   (*Предупреждение. Неисправность датчика Давления газа перед горелкой*)
   IF "P_gas_before_burner".N_module <> 0 AND "Warning_Enable".Sensor_P_gas_before_burner THEN
       "Warning".Sensor_P_gas_before_burner := "P_gas_before_burner".Error_sensor;
   ELSE
       "Warning".Sensor_P_gas_before_burner := FALSE;
   END_IF;

   (*Предупреждение. Неисправность датчика Давления воздуха к горелке*)
   IF "P_air_burner".N_module <> 0 AND "Warning_Enable".Sensor_P_air_burner THEN
       "Warning".Sensor_P_air_burner := "P_air_burner".Error_sensor;
   ELSE
       "Warning".Sensor_P_air_burner := FALSE;
   END_IF;

   (*Предупреждение. Неисправность датчика Положения рег. заслонки питательной воды на котел*)
   IF "ZRW_position".N_module <> 0 AND "Warning_Enable".Sensor_ZRW_position THEN
       "Warning".Sensor_ZRW_position := "ZRW_position".Error_sensor;
   ELSE
       "Warning".Sensor_ZRW_position := FALSE;
   END_IF;

   (*Предупреждение. Неисправность датчика Положения рег. заслонки газа перед котлом*)
   IF "ZRG_position".N_module <> 0 AND "Warning_Enable".Sensor_ZRG_position THEN
       "Warning".Sensor_ZRG_position := "ZRG_position".Error_sensor;
   ELSE
       "Warning".Sensor_ZRG_position := FALSE;
   END_IF;

   (*Предупреждение. Неисправность датчика Положения направл. аппарата вентилятора*)
   IF "NAV_position".N_module <> 0 AND "Warning_Enable".Sensor_NAV_position THEN
       "Warning".Sensor_NAV_position := "NAV_position".Error_sensor;
   ELSE
       "Warning".Sensor_NAV_position := FALSE;
   END_IF;

   (*Предупреждение. Неисправность датчика Положения направл. аппарата дымососа*)
   IF "NAD_position".N_module <> 0 AND "Warning_Enable".Sensor_NAD_position THEN
       "Warning".Sensor_NAD_position := "NAD_position".Error_sensor;
   ELSE
       "Warning".Sensor_NAD_position := FALSE;
   END_IF;

   (*Предупреждение. Неисправность датчика Температуры уходящих дымовых газов  перед экономайзером*)
   IF "T_exhaust_gas_before_economizer".N_module <> 0 AND "Warning_Enable".Sensor_T_exhaust_gas_before_economizer THEN
       "Warning".Sensor_T_exhaust_gas_before_economizer := "T_exhaust_gas_before_economizer".Error_sensor;
   ELSE
       "Warning".Sensor_T_exhaust_gas_before_economizer := FALSE;
   END_IF;

   (*Предупреждение. Неисправность датчика Температуры уходящих дымовых газов  после экономайзера*)
   IF "T_exhaust_gas_after_economizer".N_module <> 0 AND "Warning_Enable".Sensor_T_exhaust_gas_after_economizer THEN
       "Warning".Sensor_T_exhaust_gas_after_economizer := "T_exhaust_gas_after_economizer".Error_sensor;
   ELSE
       "Warning".Sensor_T_exhaust_gas_after_economizer := FALSE;
   END_IF;

   (*Предупреждение. Неисправность датчика Разрежения в дымоходе перед экономайзером*)
   IF "dP_exhaust_gas_before_economizer".N_module <> 0 AND "Warning_Enable".Sensor_dP_exhaust_gas_before_economizer THEN
       "Warning".Sensor_dP_exhaust_gas_before_economizer := "dP_exhaust_gas_before_economizer".Error_sensor;
   ELSE
       "Warning".Sensor_dP_exhaust_gas_before_economizer := FALSE;
   END_IF;

   (*Предупреждение. Неисправность датчика Разрежения в дымоходе после экономайзера*)
   IF "dP_exhaust_gas_after_economizer".N_module <> 0 AND "Warning_Enable".Sensor_dP_exhaust_gas_after_economizer THEN
       "Warning".Sensor_dP_exhaust_gas_after_economizer := "dP_exhaust_gas_after_economizer".Error_sensor;
   ELSE
       "Warning".Sensor_dP_exhaust_gas_after_economizer := FALSE;
   END_IF;

   (*Предупреждение. Неисправность датчика Уровня воды в барабане*)
   IF "L_water".N_module <> 0 AND "Warning_Enable".Sensor_L_water THEN
       "Warning".Sensor_L_water := "L_water".Error_sensor;
   ELSE
       "Warning".Sensor_L_water := FALSE;
   END_IF;

   (*Предупреждение. Неисправность датчика Давления газа перед БГ*)
   IF "P_gas_before_BG".N_module <> 0 AND "Warning_Enable".Sensor_P_gas_before_BG THEN
       "Warning".Sensor_P_gas_before_BG := "P_gas_before_BG".Error_sensor;
   ELSE
       "Warning".Sensor_P_gas_before_BG := FALSE;
   END_IF;

   (*Предупреждение. Неисправность датчика Температуры газа перед БГ*)
   IF "T_gas_before_BG".N_module <> 0 AND "Warning_Enable".Sensor_T_gas_before_BG THEN
       "Warning".Sensor_T_gas_before_BG := "T_gas_before_BG".Error_sensor;
   ELSE
       "Warning".Sensor_T_gas_before_BG := FALSE;
   END_IF;

   (*Предупреждение. Неисправность датчика Давления пара в магистраль*)
   IF "P_steam_pipe".N_module <> 0 AND "Warning_Enable".Sensor_P_steam_pipe THEN
       "Warning".Sensor_P_steam_pipe := "P_steam_pipe".Error_sensor;
   ELSE
       "Warning".Sensor_P_steam_pipe := FALSE;
   END_IF;

   (*Предупреждение. Неисправность датчика Температуры пара в магистраль*)
   IF "T_steam".N_module <> 0 AND "Warning_Enable".Sensor_T_steam THEN
       "Warning".Sensor_T_steam := "T_steam".Error_sensor;
   ELSE
       "Warning".Sensor_T_steam := FALSE;
   END_IF;

   (*Предупреждение. Неисправность датчика Текущего значение частоты ПЧ вентилятора*)
   IF "DV_current_frequency".N_module <> 0 AND "Warning_Enable".Sensor_DV_current_frequency THEN
       "Warning".Sensor_DV_current_frequency := "DV_current_frequency".Error_sensor;
   ELSE
       "Warning".Sensor_DV_current_frequency := FALSE;
   END_IF;

   (*Предупреждение. Неисправность датчика Текущего значение частоты ПЧ дымососа*)
   IF "DS_current_frequency".N_module <> 0 AND "Warning_Enable".Sensor_DS_current_frequency THEN
       "Warning".Sensor_DS_current_frequency := "DS_current_frequency".Error_sensor;
   ELSE
       "Warning".Sensor_DS_current_frequency := FALSE;
   END_IF;

   (*Предупреждение. Сработал ограничитель крутящего момента ЗДСВ перед котлом*)
   "Warning_Timer".warning_9_PT := T_CONV(INT_TO_DINT(5) * 1000);
   IF "ZDSV_before_boiler_limit_rotational_moment".Enable AND "Warning_Enable".ZDSV_before_boiler_limit_rotational_moment THEN
       "Warning_Timer".warning_9_IN := "ZDSV_before_boiler_limit_rotational_moment".Value;
       "Warning".ZDSV_before_boiler_limit_rotational_moment := "Warning_Timer".warning_9_Q;
   ELSE
       "Warning_Timer".warning_9_IN := FALSE;
       "Warning".ZDSV_before_boiler_limit_rotational_moment := FALSE;
   END_IF;

   (*Предупреждение. Сработал ограничитель крутящего момента ГПЗ*)
   "Warning_Timer".warning_10_PT := T_CONV(INT_TO_DINT(5) * 1000);
   IF "GPZ_limit_rotational_moment".Enable AND "Warning_Enable".GPZ_limit_rotational_moment THEN
       "Warning_Timer".warning_10_IN := "GPZ_limit_rotational_moment".Value;
       "Warning".GPZ_limit_rotational_moment := "Warning_Timer".warning_10_Q;
   ELSE
       "Warning_Timer".warning_10_IN := FALSE;
       "Warning".GPZ_limit_rotational_moment := FALSE;
   END_IF;

   (*Предупреждение. Вызов к шакафу электропитания*)
   IF "Call_power_supply_cabinet".N_module<>0 AND "Warning_Enable".Call_power_supply_cabinet THEN
       "Warning".Call_power_supply_cabinet := "Call_power_supply_cabinet".Value;
   ELSE
       "Warning".Call_power_supply_cabinet := FALSE;
   END_IF;

   (*Предупреждение. ДВ. Необходимо включить QF ПЧ*)
   IF "DV_dist_control".Value AND "DV_invertor_mode".Value AND NOT "DV_invertor_QF_on".Value AND "DV_invertor_QF_on".N_module<>0 AND "Warning_Enable".DV_need_on_QF_invertor THEN
       "Warning".DV_need_on_QF_invertor := TRUE;
   ELSE
       "Warning".DV_need_on_QF_invertor := FALSE;
   END_IF;

   (*Предупреждение. ДВ. Необходимо включить QF Сети*)
   IF "DV_dist_control".Value AND "DV_powergrid_mode".Value AND NOT "DV_powergrid_QF_on".Value AND "DV_powergrid_QF_on".N_module<>0 AND "Warning_Enable".DV_need_on_QF_powergrid THEN
       "Warning".DV_need_on_QF_powergrid := TRUE;
   ELSE
       "Warning".DV_need_on_QF_powergrid := FALSE;
   END_IF;

   (*Предупреждение. ДВ. Неисправность напряжения в Сети ШУД*)
   IF "DV_no_voltage".N_module<>0 AND "Warning_Enable".DV_no_voltage THEN
       "Warning".DV_no_voltage := "DV_no_voltage".Value;
   ELSE
       "Warning".DV_no_voltage := FALSE;
   END_IF;

   (*Предупреждение. ДС. Необходимо включить QF ПЧ*)
   IF "DS_dist_control".Value AND "DS_invertor_mode".Value AND NOT "DS_invertor_QF_on".Value AND "DS_invertor_QF_on".N_module<>0 AND "Warning_Enable".DS_need_on_QF_invertor THEN
       "Warning".DS_need_on_QF_invertor := TRUE;
   ELSE
       "Warning".DS_need_on_QF_invertor := FALSE;
   END_IF;

   (*Предупреждение. ДС. Необходимо включить QF Сети*)
   IF "DS_dist_control".Value AND "DS_powergrid_mode".Value AND NOT "DS_powergrid_QF_on".Value AND "DS_powergrid_QF_on".N_module<>0 AND "Warning_Enable".DS_need_on_QF_powergrid THEN
       "Warning".DS_need_on_QF_powergrid := TRUE;
   ELSE
       "Warning".DS_need_on_QF_powergrid := FALSE;
   END_IF;

   (*Предупреждение. ДС. Неисправность напряжения в Сети ШУД*)
   IF "DS_no_voltage".N_module<>0 AND "Warning_Enable".DS_no_voltage THEN
       "Warning".DS_no_voltage := "DS_no_voltage".Value;
   ELSE
       "Warning".DS_no_voltage := FALSE;
   END_IF;

   (*Предупреждение. Нет питания ШЭУ*)
   IF "SHEU_voltage_ok".N_module<>0 AND "Warning_Enable".SHEU_no_voltage THEN
       "Warning".SHEU_no_voltage := NOT "SHEU_voltage_ok".Value;
   ELSE
       "Warning".SHEU_no_voltage := FALSE;
   END_IF;

   (*Предупреждение. Питание контроллера от ИБП*)
   IF "Power_PLC_from_UPS".N_module<>0 AND "Warning_Enable".Power_PLC_from_UPS THEN
       "Warning".Power_PLC_from_UPS := "Power_PLC_from_UPS".Value;
   ELSE
       "Warning".Power_PLC_from_UPS := FALSE;
   END_IF;

   (*Предупреждение. Низкий заряд батареи ИБП*)
   IF "UPS_Low_charge".N_module<>0 AND "Warning_Enable".UPS_Low_charge THEN
       "Warning".UPS_Low_charge := "UPS_Low_charge".Value;
   ELSE
       "Warning".UPS_Low_charge := FALSE;
   END_IF;

   (*Предупреждение. Нет питания ЗРГ*)
   IF "ZRG_voltage_ok".N_module<>0 AND "Warning_Enable".ZRG_no_voltage THEN
       "Warning".ZRG_no_voltage := NOT "ZRG_voltage_ok".Value;
   ELSE
       "Warning".ZRG_no_voltage := FALSE;
   END_IF;

   (*Предупреждение. Нет питания ЗДГ*)
   IF "ZDG_voltage_ok".N_module<>0 AND "Warning_Enable".ZDG_no_voltage THEN
       "Warning".ZDG_no_voltage := NOT "ZDG_voltage_ok".Value;
   ELSE
       "Warning".ZDG_no_voltage := FALSE;
   END_IF;

   (*Предупреждение. Нет питания НАВ*)
   IF "NAV_voltage_ok".N_module<>0 AND "Warning_Enable".NAV_no_voltage THEN
       "Warning".NAV_no_voltage := NOT "NAV_voltage_ok".Value;
   ELSE
       "Warning".NAV_no_voltage := FALSE;
   END_IF;

   (*Предупреждение. Нет питания НАД*)
   IF "NAD_voltage_ok".N_module<>0 AND "Warning_Enable".NAD_no_voltage THEN
       "Warning".NAD_no_voltage := NOT "NAD_voltage_ok".Value;
   ELSE
       "Warning".NAD_no_voltage := FALSE;
   END_IF;

   (*Предупреждение. Нет питания ЗДСВ перед котлом*)
   IF "ZDSV_before_boiler_voltage_ok".N_module<>0 AND "Warning_Enable".ZDSV_before_boiler_no_voltage THEN
       "Warning".ZDSV_before_boiler_no_voltage := NOT "ZDSV_before_boiler_voltage_ok".Value;
   ELSE
       "Warning".ZDSV_before_boiler_no_voltage := FALSE;
   END_IF;

   (*Предупреждение. Нет питания ГПЗ*)
   IF "GPZ_voltage_ok".N_module <> 0 AND "Warning_Enable".GPZ_no_voltage THEN
       "Warning".GPZ_no_voltage := NOT "GPZ_voltage_ok".Value;
   ELSE
       "Warning".GPZ_no_voltage := FALSE;
   END_IF;

   (*Предупреждение. Нет питания ЗРВ*)
   IF "ZRW_voltage_ok".N_module <> 0 AND "Warning_Enable".ZRW_no_voltage THEN
       "Warning".ZRW_no_voltage := NOT "ZRW_voltage_ok".Value;
   ELSE
       "Warning".ZRW_no_voltage := FALSE;
   END_IF;

   (*Предупреждение. Авария ПЧ ДВ*)
   IF "DV_Invertor_alarm".N_module<>0 AND "DV_invertor_mode".Value AND "Warning_Enable".DV_invertor_alarm THEN
       "Warning".DV_invertor_alarm := "DV_Invertor_alarm".Value;
   ELSE
       "Warning".DV_invertor_alarm := FALSE;
   END_IF;

   (*Предупреждение. Авария ПЧ ДС*)
   IF "DS_Invertor_alarm".N_module<>0 AND "DS_invertor_mode".Value AND "Warning_Enable".DS_invertor_alarm THEN
       "Warning".DS_invertor_alarm := "DS_Invertor_alarm".Value;
   ELSE
       "Warning".DS_invertor_alarm := FALSE;
   END_IF;

   (*Предупреждение. ЗРГ в местном режиме управления*)
   "Warning".ZRG_manual := "Warning_Enable".ZRG_manual AND NOT "ZRG_avto".Value;

   (*Предупреждение. НАВ в местном режиме управления*)
   "Warning".NAV_manual := "Warning_Enable".NAV_manual AND NOT "NAV_avto".Value;

   (*Предупреждение. НАД в местном режиме управления*)
   "Warning".NAD_manual := "Warning_Enable".NAD_manual AND NOT "NAD_avto".Value;

   (*Предупреждение. ДВ в местном режиме управления*)
   "Warning".DV_manual := "Warning_Enable".DV_manual AND "DV_local_control".Value;

   (*Предупреждение. ДС в местном режиме управления*)
   "Warning".DS_manual := "Warning_Enable".DS_manual AND "DS_local_control".Value;

   (*Предупреждение. ЗРВ в местном режиме управления*)
   "Warning".ZRW_manual := "Warning_Enable".ZRW_manual AND NOT "ZRW_avto".Value;

   (*Пламя запальника потухло*)
   "Warning_Timer".warning_1_PT := T_CONV(INT_TO_DINT("Warning_SP".TIME_Not_flame_Igniter));
   IF "Warning_Enable".Not_flame_Igniter THEN
       "Warning_Timer".warning_1_IN := NOT "Igniter_flame".Value;
       IF "Warning_Timer".warning_1_Q THEN
           "Warning".Not_flame_Igniter := TRUE;
       END_IF;
   ELSE
       "Warning_Timer".warning_1_IN := FALSE;
       //"Warning".Not_flame_Igniter := FALSE;
   END_IF;

   (*ПЗК2 не открылся*)
   "Warning_Timer".warning_2_PT := T_CONV(INT_TO_DINT("Warning_SP".TIME_PZK2_not_open) * 1000);
   IF "Warning_Enable".PZK2_not_open THEN
       "Warning_Timer".warning_2_IN := NOT "PZK2_open".Value;
       IF "Warning_Timer".warning_2_Q THEN
           "Warning".PZK2_not_open := TRUE;
       END_IF;
   ELSE
       "Warning_Timer".warning_2_IN := FALSE;
       //"Warning".PZK2_not_open := FALSE;
   END_IF;

   (*Понижение давления сетевой воды*)
   IF ("P_water_before_regul".Value <"Warning_SP".P_water_min AND NOT"P_water_before_regul".Error_sensor AND "P_water_before_regul".N_module <> 0) THEN
       "Warning".P_water_min := TRUE;
   ELSE
       "Warning".P_water_min := FALSE;
   END_IF;

   (*Понижение уровня воды в барабане*)
   "Warning_Timer".warning_3_PT := T_CONV(INT_TO_DINT("Warning_SP".TIME_L_water_min) * 1000);
   IF "Warning_Enable".L_water_min THEN
       "Warning_Timer".warning_3_IN := "L_water".Value < "Warning_SP".L_water_min AND NOT "L_water".Error_sensor AND "L_water".N_module <> 0;
       "Warning".L_water_min := "Warning_Timer".warning_3_Q;
   ELSE
       "Warning_Timer".warning_3_IN := FALSE;
       "Warning".L_water_min := FALSE;
   END_IF;

   (*Повышение уровня воды в барабане*)
   "Warning_Timer".warning_4_PT := T_CONV(INT_TO_DINT("Warning_SP".TIME_L_water_max) * 1000);
   IF "Warning_Enable".L_water_max THEN
       "Warning_Timer".warning_4_IN := "L_water".Value > "Warning_SP".L_water_max AND NOT "L_water".Error_sensor AND "L_water".N_module <> 0;
       "Warning".L_water_max := "Warning_Timer".warning_4_Q;
   ELSE
       "Warning_Timer".warning_4_IN := FALSE;
       "Warning".L_water_max := FALSE;
   END_IF;

   (*Повышение давления пара в барабане*)
   "Warning_Timer".warning_5_PT := T_CONV(INT_TO_DINT("Warning_SP".TIME_P_steam_max) * 1000);
   IF "Warning_Enable".P_steam_max THEN
       "Warning_Timer".warning_5_IN := "P_steam".Value > "Warning_SP".P_steam_max AND NOT "P_steam".Error_sensor AND "P_steam".N_module <> 0;
       "Warning".P_steam_max := "Warning_Timer".warning_5_Q;
   ELSE
       "Warning_Timer".warning_5_IN := FALSE;
       "Warning".P_steam_max := FALSE;
   END_IF;

   (*СО порог 1*)
   IF "Warning_Enable".CO2 THEN
       "Warning".CO2 := "CO_1".Value;
   ELSE
       "Warning".CO2 := FALSE;
   END_IF;

   (*Предупреждение. Понижение разряжения в топке*)
   "Warning_Timer".warning_6_PT := T_CONV(INT_TO_DINT("Alarm_SP".TIME_dP_furnace_boiler_min) * 1000);
   IF "Technology".Regim = 3 AND ("Technology".Regim_ventilation_step = 23 OR "Technology".Regim_ventilation_step = 24) AND "Warning_Enable".dP_furnace_boiler_min THEN
       "Warning_Timer".warning_6_IN := "dP_furnace_boiler_min".Value OR ("dP_furnace_boiler".Value > "Alarm_SP".dP_furnace_boiler_min AND NOT "dP_furnace_boiler".Error_sensor AND "dP_furnace_boiler".N_module <> 0);
       IF "Warning_Timer".warning_6_Q THEN
           "Warning".dP_furnace_boiler_min := TRUE;
       END_IF;
   ELSE
       "Warning_Timer".warning_6_IN := FALSE;
       "Warning".dP_furnace_boiler_min := FALSE;
   END_IF;

   (*Предупреждение. Понижение давления воздуха перед горелкой *)
   "Warning_Timer".warning_7_PT := T_CONV(INT_TO_DINT("Alarm_SP".TIME_P_air_before_burner_min) * 1000);
   IF "Technology".Regim = 3 AND ("Technology".Regim_ventilation_step = 23 OR "Technology".Regim_ventilation_step = 24) AND "Warning_Enable".P_air_before_burner_min THEN
       "Warning_Timer".warning_7_IN := "P_air_before_burner_min".Value OR ("P_air_burner".Value < "Alarm_SP".P_air_before_burner_min AND NOT "P_air_burner".Error_sensor AND "P_air_burner".N_module<>0);
       IF "Warning_Timer".warning_7_Q THEN
           "Warning".P_air_before_burner_min := TRUE;
       END_IF;
   ELSE
       "Warning_Timer".warning_7_IN := FALSE;
       "Warning".P_air_before_burner_min := FALSE;
   END_IF;

   (*ЗДГ не закрылась*)
   "Warning_Timer".warning_8_PT := T_CONV(INT_TO_DINT("Warning_SP".TIME_ZDG_not_close) * 1000);
   IF "Warning_Enable".ZDG_not_close THEN
       "Warning_Timer".warning_8_IN := "ZDG_no_close".Value;
       IF "Warning_Timer".warning_8_Q THEN
           "Warning".ZDG_not_close := TRUE;
       END_IF;
   ELSE
       "Warning_Timer".warning_8_IN := FALSE;
   END_IF;

   (*Предупреждение. Имеется блокировка защиты *)
   IF "Protections_BLOCK".P_gas_before_BG_max OR
       "Protections_BLOCK".P_gas_before_BG_min OR
       "Protections_BLOCK".P_gas_before_burner_min OR
       "Protections_BLOCK".P_gas_before_burner_max OR
       "Protections_BLOCK".DS_off OR
       "Protections_BLOCK".DV_off OR
       "Protections_BLOCK".dP_in_furnance_min OR
       "Protections_BLOCK".P_air_before_burner_min OR
       "Protections_BLOCK".L_water_min OR
       "Protections_BLOCK".L_water_max OR
       "Protections_BLOCK".P_steam_max OR
       "Protections_BLOCK".Not_flame_burner OR
       "Protections_BLOCK".Alarm_stop_HMI OR
       "Protections_BLOCK".Alarm_stop_SCADA THEN
       "Warning".protection_block := TRUE;
   ELSE
       "Warning".protection_block := FALSE;
   END_IF;

   (*СБРОС аварий для журнала событий*)
   IF "Alarm".Reset_alarms THEN
       "HMI".Reset_alarms_Log := TRUE;
   END_IF;

   (*Сброс всех аварий и предупреждений*)
   IF "Alarm".Reset_alarms = TRUE OR
       "Btn_Sound".Value THEN
       (*Повышение давления газа перед БГ*)
       IF NOT "Alarm_Timer".alarm_1_Q THEN
           "Alarm".P_gas_before_BG_max := FALSE;
       END_IF;
       (*Понижение давления газа перед БГ*)
       IF NOT "Alarm_Timer".alarm_2_Q THEN
           "Alarm".P_gas_before_BG_min := FALSE;
       END_IF;
       (*Понижение давления газа перед горелкой*)
       IF NOT "Alarm_Timer".alarm_3_Q THEN
           "Alarm".P_gas_before_burner_min := FALSE;
       END_IF;
       (*Повышение давления газа перед горелкой*)
       IF NOT "Alarm_Timer".alarm_4_Q THEN
           "Alarm".P_gas_before_burner_max := FALSE;
       END_IF;
       (*Отключение ДС*)
       IF NOT "Alarm_Timer".alarm_5_Q THEN
           "Alarm".DS_off := FALSE;
       END_IF;
       (*Отключение ДВ*)
       IF NOT "Alarm_Timer".alarm_6_Q THEN
           "Alarm".DV_off := FALSE;
       END_IF;
       (*Понижение разряжения в топке*)
       IF NOT "Alarm_Timer".alarm_7_Q THEN
           "Alarm".dP_furnace_boiler_min := FALSE;
       END_IF;
       (*Понижение давления воздуха перед горелкой *)
       IF NOT "Alarm_Timer".alarm_8_Q THEN
           "Alarm".P_air_before_burner_min := FALSE;
       END_IF;
       (*Понижение уровня воды в барабане*)
       IF NOT "Alarm_Timer".alarm_9_Q THEN
           "Alarm".L_water_min := FALSE;
       END_IF;
       (*Повышение уровня воды в барабане*)
       IF NOT "Alarm_Timer".alarm_10_Q THEN
           "Alarm".L_water_max := FALSE;
       END_IF;
       (*Повышение давления пара в барабане*)
       IF NOT "Alarm_Timer".alarm_11_Q THEN
           "Alarm".P_steam_max := FALSE;
       END_IF;
       (*Невоспламенение или погасание факела горелки котла*)
       IF NOT "Alarm_Timer".alarm_12_Q THEN
           "Alarm".Not_flame_burner := FALSE;
       END_IF;
       (*Нажата кнопка аварийного останова на панели оператора*)
       "Alarm".Alarm_stop_HMI := FALSE;
       (*Нажата кнопка аварийного останова на SCADA*)
       "Alarm".Alarm_stop_SCADA := FALSE;
       (*СО2 порог 2*)
       IF NOT "Alarm_Timer".alarm_13_Q THEN
           "Alarm".CO2 := FALSE;
       END_IF;
       (*CH4*)
       IF NOT "Alarm_Timer".alarm_14_Q THEN
           "Alarm".CH4 := FALSE;
       END_IF;
       (*Пламя запальника потухло*)
       IF NOT "Warning_Timer".warning_1_Q THEN
           "Warning".Not_flame_Igniter := FALSE;
       END_IF;
       (*ПЗК2 не открылся*)
       IF NOT "Warning_Timer".warning_2_Q THEN
           "Warning".PZK2_not_open := FALSE;
       END_IF;
       (*Понижение уровня воды в барабане*)
       IF NOT "Warning_Timer".warning_3_Q THEN
           "Warning".L_water_min := FALSE;
       END_IF;
       (*Повышение уровня воды в барабане*)
       IF NOT "Warning_Timer".warning_4_Q THEN
           "Warning".L_water_max := FALSE;
       END_IF;
       (*Повышение давления пара в барабане*)
       IF NOT "Warning_Timer".warning_5_Q THEN
           "Warning".P_steam_max := FALSE;
       END_IF;
       (*Предупреждение. Понижение разряжения в топке*)
       IF NOT "Warning_Timer".warning_6_Q THEN
           "Warning".dP_furnace_boiler_min := FALSE;
       END_IF;
       (*Предупреждение. Понижение давления воздуха перед горелкой *)
       IF NOT "Warning_Timer".warning_7_Q THEN
           "Warning".P_air_before_burner_min := FALSE;
       END_IF;
       (*ЗДГ не закрылась*)
       IF NOT "Warning_Timer".warning_8_Q THEN
           "Warning".ZDG_not_close := FALSE;
       END_IF;
       "Alarm".Reset_alarms := FALSE;
   END_IF;

   (*Формирование обобщенного признака аварии*)
   "Alarm".Global_alarm := "Alarm".P_gas_before_BG_max OR
   "Alarm".P_gas_before_BG_min OR
   "Alarm".P_gas_before_burner_min OR
   "Alarm".P_gas_before_burner_max OR
   "Alarm".DS_off OR
   "Alarm".DV_off OR
   "Alarm".dP_furnace_boiler_min OR
   "Alarm".P_air_before_burner_min OR
   "Alarm".L_water_min OR
   "Alarm".L_water_max OR
   "Alarm".P_steam_max OR
   "Alarm".Not_flame_burner OR
   "Alarm".Alarm_stop_HMI OR
   "Alarm".Alarm_stop_SCADA OR
   "Alarm".CO2 OR
   "Alarm".CH4;

   (*ловим передний фронт аварий*) 
   "R_TRIG_DB_alarm1"(CLK :="Alarm".P_gas_before_BG_max,
                      Q =>"FRONT".Alarm_1);
   "R_TRIG_DB_alarm2"(CLK :="Alarm".P_gas_before_BG_min,
                      Q =>"FRONT".Alarm_2);
   "R_TRIG_DB_alarm3"(CLK :="Alarm".P_gas_before_burner_min,
                      Q =>"FRONT".Alarm_3);
   "R_TRIG_DB_alarm4"(CLK :="Alarm".P_gas_before_burner_max,
                      Q =>"FRONT".Alarm_4);
   "R_TRIG_DB_alarm5"(CLK :="Alarm".DS_off,
                      Q =>"FRONT".Alarm_5);
   "R_TRIG_DB_alarm6"(CLK :="Alarm".DV_off,
                      Q =>"FRONT".Alarm_6);
   "R_TRIG_DB_alarm7"(CLK :="Alarm".dP_furnace_boiler_min,
                      Q =>"FRONT".Alarm_7);
   "R_TRIG_DB_alarm8"(CLK := "Alarm".P_air_before_burner_min,
                      Q =>"FRONT".Alarm_8);
   "R_TRIG_DB_alarm9"(CLK :="Alarm".L_water_min,
                      Q =>"FRONT".Alarm_9);
   "R_TRIG_DB_alarm10"(CLK :="Alarm".L_water_max,
                       Q =>"FRONT".Alarm_10);
   "R_TRIG_DB_alarm11"(CLK :="Alarm".P_steam_max,
                       Q =>"FRONT".Alarm_11);
   "R_TRIG_DB_alarm12"(CLK :="Alarm".Not_flame_burner,
                       Q =>"FRONT".Alarm_12);
   "R_TRIG_DB_alarm13"(CLK :="Alarm".Alarm_stop_HMI,
                       Q =>"FRONT".Alarm_13);
   "R_TRIG_DB_alarm14"(CLK :="Alarm".Alarm_stop_SCADA,
                       Q =>"FRONT".Alarm_14);
   "R_TRIG_DB_alarm15"(CLK :="Alarm".CO2,
                       Q =>"FRONT".Alarm_15);
   "R_TRIG_DB_alarm16"(CLK :="Alarm".CH4,
                       Q =>"FRONT".Alarm_16);

   "TON_test_sound_DB".TON(IN := "Timer".test_sound_IN,
   PT := "Timer".test_sound_PT,
   Q => "Timer".test_sound_Q);

   (*Управление звуковой сигнализацией*)
   "Timer".test_sound_PT := T#2s;
   "Timer".test_sound_IN := "Btn_Sound".Value;
   IF "FRONT".Alarm_1 OR
       "FRONT".Alarm_2 OR
       "FRONT".Alarm_3 OR
       "FRONT".Alarm_4 OR
       "FRONT".Alarm_5 OR
       "FRONT".Alarm_6 OR
       "FRONT".Alarm_7 OR
       "FRONT".Alarm_8 OR
       "FRONT".Alarm_9 OR
       "FRONT".Alarm_10 OR
       "FRONT".Alarm_11 OR
       "FRONT".Alarm_12 OR
       "FRONT".Alarm_13 OR
       "FRONT".Alarm_14 OR
       "FRONT".Alarm_15 OR
       "FRONT".Alarm_16 OR
       "Timer".test_sound_Q THEN
       "control_alarm_signal".Value := TRUE;
   ELSE
       //отключение звуковой сигнализации
       IF (NOT "Alarm".Global_alarm AND NOT "Timer".test_sound_Q) OR "FRONT".Btn_reset_sound_HMI THEN
           "control_alarm_signal".Value := FALSE;
       END_IF;
   END_IF;
END_FUNCTION

FUNCTION "write_discret" : Void   // FC6, SCL
{ S7_Optimized_Access := 'TRUE' }
AUTHOR : Dmitriy_Petrov
VERSION : 0.1
// Функция записи дискретного параметра
   VAR_INPUT
      Value : Bool;   // Значение сигнала
      Invert : Bool;   // Инвертирование сигнала
   END_VAR
   VAR_IN_OUT
      N_module : USInt;   // № модуля (начиная с 1)
      N_chanel : USInt;   // № канала (начиная с 1)
   END_VAR
   VAR_TEMP
      Signal : Bool;   // Значение сигнала для записи
   END_VAR
BEGIN
   (*проверка правильности введеного значения № Модуля*)
   IF #N_module < 1 OR #N_module > 25 THEN
       #N_module := 0;
   END_IF;

   (*проверка правильности введеного значения № Канала*)
   IF #N_module = 0 THEN
       #N_chanel := 0;
   ELSE
       IF #N_chanel < 1 OR #N_chanel > 16 THEN
           #N_chanel := 0;
       END_IF;
   END_IF;

   (*инвертирование сигнала (при необходимости)*)
   IF NOT #Invert THEN
       #Signal := #Value;
   ELSE
       #Signal := NOT #Value;
   END_IF;

   (*запись дискретного сигнала в выбранный канал*)
   CASE #N_module OF
       1:  // Модуль 1
           CASE #N_chanel OF
               1:
                   "Module01Chanel1_DO" := #Signal;   //Канал 1
               2:
                   "Module01Chanel2_DO" := #Signal;   //Канал 2
               3:
                   "Module01Chanel3_DO" := #Signal;   //Канал 3
               4:
                   "Module01Chanel4_DO" := #Signal;   //Канал 4
               5:
                   "Module01Chanel5_DO" := #Signal;   //Канал 5
               6:
                   "Module01Chanel6_DO" := #Signal;   //Канал 6
               7:
                   "Module01Chanel7_DO" := #Signal;   //Канал 7
               8:
                   "Module01Chanel8_DO" := #Signal;   //Канал 8
               9:
                   "Module01Chanel9_DO" := #Signal;   //Канал 9
               10:
                   "Module01Chanel10_DO" := #Signal;   //Канал 10
               11:
                   "Module01Chanel11_DO" := #Signal;   //Канал 11
               12:
                   "Module01Chanel12_DO" := #Signal;   //Канал 12
               13:
                   "Module01Chanel13_DO" := #Signal;   //Канал 13
               14:
                   "Module01Chanel14_DO" := #Signal;   //Канал 14
               15:
                   "Module01Chanel15_DO" := #Signal;   //Канал 15
               16:
                   "Module01Chanel16_DO" := #Signal;   //Канал 16
           END_CASE;
       2:  // Модуль 2
           CASE #N_chanel OF
               1:
                   "Module02Chanel1_DO" := #Signal;   //Канал 1
               2:
                   "Module02Chanel2_DO" := #Signal;   //Канал 2
               3:
                   "Module02Chanel3_DO" := #Signal;   //Канал 3
               4:
                   "Module02Chanel4_DO" := #Signal;   //Канал 4
               5:
                   "Module02Chanel5_DO" := #Signal;   //Канал 5
               6:
                   "Module02Chanel6_DO" := #Signal;   //Канал 6
               7:
                   "Module02Chanel7_DO" := #Signal;   //Канал 7
               8:
                   "Module02Chanel8_DO" := #Signal;   //Канал 8
               9:
                   "Module02Chanel9_DO" := #Signal;   //Канал 9
               10:
                   "Module02Chanel10_DO" := #Signal;   //Канал 10
               11:
                   "Module02Chanel11_DO" := #Signal;   //Канал 11
               12:
                   "Module02Chanel12_DO" := #Signal;   //Канал 12
               13:
                   "Module02Chanel13_DO" := #Signal;   //Канал 13
               14:
                   "Module02Chanel14_DO" := #Signal;   //Канал 14
               15:
                   "Module02Chanel15_DO" := #Signal;   //Канал 15
               16:
                   "Module02Chanel16_DO" := #Signal;   //Канал 16
           END_CASE;
       3:  // Модуль 3
           CASE #N_chanel OF
               1:
                   "Module03Chanel1_DO" := #Signal;   //Канал 1
               2:
                   "Module03Chanel2_DO" := #Signal;   //Канал 2
               3:
                   "Module03Chanel3_DO" := #Signal;   //Канал 3
               4:
                   "Module03Chanel4_DO" := #Signal;   //Канал 4
               5:
                   "Module03Chanel5_DO" := #Signal;   //Канал 5
               6:
                   "Module03Chanel6_DO" := #Signal;   //Канал 6
               7:
                   "Module03Chanel7_DO" := #Signal;   //Канал 7
               8:
                   "Module03Chanel8_DO" := #Signal;   //Канал 8
               9:
                   "Module03Chanel9_DO" := #Signal;   //Канал 9
               10:
                   "Module03Chanel10_DO" := #Signal;   //Канал 10
               11:
                   "Module03Chanel11_DO" := #Signal;   //Канал 11
               12:
                   "Module03Chanel12_DO" := #Signal;   //Канал 12
               13:
                   "Module03Chanel13_DO" := #Signal;   //Канал 13
               14:
                   "Module03Chanel14_DO" := #Signal;   //Канал 14
               15:
                   "Module03Chanel15_DO" := #Signal;   //Канал 15
               16:
                   "Module03Chanel16_DO" := #Signal;   //Канал 16
           END_CASE;
       4:  // Модуль 4
           CASE #N_chanel OF
               1:
                   "Module04Chanel1_DO" := #Signal;   //Канал 1
               2:
                   "Module04Chanel2_DO" := #Signal;   //Канал 2
               3:
                   "Module04Chanel3_DO" := #Signal;   //Канал 3
               4:
                   "Module04Chanel4_DO" := #Signal;   //Канал 4
               5:
                   "Module04Chanel5_DO" := #Signal;   //Канал 5
               6:
                   "Module04Chanel6_DO" := #Signal;   //Канал 6
               7:
                   "Module04Chanel7_DO" := #Signal;   //Канал 7
               8:
                   "Module04Chanel8_DO" := #Signal;   //Канал 8
               9:
                   "Module04Chanel9_DO" := #Signal;   //Канал 9
               10:
                   "Module04Chanel10_DO" := #Signal;   //Канал 10
               11:
                   "Module04Chanel11_DO" := #Signal;   //Канал 11
               12:
                   "Module04Chanel12_DO" := #Signal;   //Канал 12
               13:
                   "Module04Chanel13_DO" := #Signal;   //Канал 13
               14:
                   "Module04Chanel14_DO" := #Signal;   //Канал 14
               15:
                   "Module04Chanel15_DO" := #Signal;   //Канал 15
               16:
                   "Module04Chanel16_DO" := #Signal;   //Канал 16
           END_CASE;
       5:  // Модуль 5
           CASE #N_chanel OF
               1:
                   "Module05Chanel1_DO" := #Signal;   //Канал 1
               2:
                   "Module05Chanel2_DO" := #Signal;   //Канал 2
               3:
                   "Module05Chanel3_DO" := #Signal;   //Канал 3
               4:
                   "Module05Chanel4_DO" := #Signal;   //Канал 4
               5:
                   "Module05Chanel5_DO" := #Signal;   //Канал 5
               6:
                   "Module05Chanel6_DO" := #Signal;   //Канал 6
               7:
                   "Module05Chanel7_DO" := #Signal;   //Канал 7
               8:
                   "Module05Chanel8_DO" := #Signal;   //Канал 8
               9:
                   "Module05Chanel9_DO" := #Signal;   //Канал 9
               10:
                   "Module05Chanel10_DO" := #Signal;   //Канал 10
               11:
                   "Module05Chanel11_DO" := #Signal;   //Канал 11
               12:
                   "Module05Chanel12_DO" := #Signal;   //Канал 12
               13:
                   "Module05Chanel13_DO" := #Signal;   //Канал 13
               14:
                   "Module05Chanel14_DO" := #Signal;   //Канал 14
               15:
                   "Module05Chanel15_DO" := #Signal;   //Канал 15
               16:
                   "Module05Chanel16_DO" := #Signal;   //Канал 16
           END_CASE;
       6:  // Модуль 6
           CASE #N_chanel OF
               1:
                   "Module06Chanel1_DO" := #Signal;   //Канал 1
               2:
                   "Module06Chanel2_DO" := #Signal;   //Канал 2
               3:
                   "Module06Chanel3_DO" := #Signal;   //Канал 3
               4:
                   "Module06Chanel4_DO" := #Signal;   //Канал 4
               5:
                   "Module06Chanel5_DO" := #Signal;   //Канал 5
               6:
                   "Module06Chanel6_DO" := #Signal;   //Канал 6
               7:
                   "Module06Chanel7_DO" := #Signal;   //Канал 7
               8:
                   "Module06Chanel8_DO" := #Signal;   //Канал 8
               9:
                   "Module06Chanel9_DO" := #Signal;   //Канал 9
               10:
                   "Module06Chanel10_DO" := #Signal;   //Канал 10
               11:
                   "Module06Chanel11_DO" := #Signal;   //Канал 11
               12:
                   "Module06Chanel12_DO" := #Signal;   //Канал 12
               13:
                   "Module06Chanel13_DO" := #Signal;   //Канал 13
               14:
                   "Module06Chanel14_DO" := #Signal;   //Канал 14
               15:
                   "Module06Chanel15_DO" := #Signal;   //Канал 15
               16:
                   "Module06Chanel16_DO" := #Signal;   //Канал 16
           END_CASE;
       7:  // Модуль 7
           CASE #N_chanel OF
               1:
                   "Module07Chanel1_DO" := #Signal;   //Канал 1
               2:
                   "Module07Chanel2_DO" := #Signal;   //Канал 2
               3:
                   "Module07Chanel3_DO" := #Signal;   //Канал 3
               4:
                   "Module07Chanel4_DO" := #Signal;   //Канал 4
               5:
                   "Module07Chanel5_DO" := #Signal;   //Канал 5
               6:
                   "Module07Chanel6_DO" := #Signal;   //Канал 6
               7:
                   "Module07Chanel7_DO" := #Signal;   //Канал 7
               8:
                   "Module07Chanel8_DO" := #Signal;   //Канал 8
               9:
                   "Module07Chanel9_DO" := #Signal;   //Канал 9
               10:
                   "Module07Chanel10_DO" := #Signal;   //Канал 10
               11:
                   "Module07Chanel11_DO" := #Signal;   //Канал 11
               12:
                   "Module07Chanel12_DO" := #Signal;   //Канал 12
               13:
                   "Module07Chanel13_DO" := #Signal;   //Канал 13
               14:
                   "Module07Chanel14_DO" := #Signal;   //Канал 14
               15:
                   "Module07Chanel15_DO" := #Signal;   //Канал 15
               16:
                   "Module07Chanel16_DO" := #Signal;   //Канал 16
           END_CASE;
       8:  // Модуль 8
           CASE #N_chanel OF
               1:
                   "Module08Chanel1_DO" := #Signal;   //Канал 1
               2:
                   "Module08Chanel2_DO" := #Signal;   //Канал 2
               3:
                   "Module08Chanel3_DO" := #Signal;   //Канал 3
               4:
                   "Module08Chanel4_DO" := #Signal;   //Канал 4
               5:
                   "Module08Chanel5_DO" := #Signal;   //Канал 5
               6:
                   "Module08Chanel6_DO" := #Signal;   //Канал 6
               7:
                   "Module08Chanel7_DO" := #Signal;   //Канал 7
               8:
                   "Module08Chanel8_DO" := #Signal;   //Канал 8
               9:
                   "Module08Chanel9_DO" := #Signal;   //Канал 9
               10:
                   "Module08Chanel10_DO" := #Signal;   //Канал 10
               11:
                   "Module08Chanel11_DO" := #Signal;   //Канал 11
               12:
                   "Module08Chanel12_DO" := #Signal;   //Канал 12
               13:
                   "Module08Chanel13_DO" := #Signal;   //Канал 13
               14:
                   "Module08Chanel14_DO" := #Signal;   //Канал 14
               15:
                   "Module08Chanel15_DO" := #Signal;   //Канал 15
               16:
                   "Module08Chanel16_DO" := #Signal;   //Канал 16
           END_CASE;
       9:  // Модуль 9
           CASE #N_chanel OF
               1:
                   "Module09Chanel1_DO" := #Signal;   //Канал 1
               2:
                   "Module09Chanel2_DO" := #Signal;   //Канал 2
               3:
                   "Module09Chanel3_DO" := #Signal;   //Канал 3
               4:
                   "Module09Chanel4_DO" := #Signal;   //Канал 4
               5:
                   "Module09Chanel5_DO" := #Signal;   //Канал 5
               6:
                   "Module09Chanel6_DO" := #Signal;   //Канал 6
               7:
                   "Module09Chanel7_DO" := #Signal;   //Канал 7
               8:
                   "Module09Chanel8_DO" := #Signal;   //Канал 8
               9:
                   "Module09Chanel9_DO" := #Signal;   //Канал 9
               10:
                   "Module09Chanel10_DO" := #Signal;   //Канал 10
               11:
                   "Module09Chanel11_DO" := #Signal;   //Канал 11
               12:
                   "Module09Chanel12_DO" := #Signal;   //Канал 12
               13:
                   "Module09Chanel13_DO" := #Signal;   //Канал 13
               14:
                   "Module09Chanel14_DO" := #Signal;   //Канал 14
               15:
                   "Module09Chanel15_DO" := #Signal;   //Канал 15
               16:
                   "Module09Chanel16_DO" := #Signal;   //Канал 16
           END_CASE;
       10:  // Модуль 10
           CASE #N_chanel OF
               1:
                   "Module10Chanel1_DO" := #Signal;   //Канал 1
               2:
                   "Module10Chanel2_DO" := #Signal;   //Канал 2
               3:
                   "Module10Chanel3_DO" := #Signal;   //Канал 3
               4:
                   "Module10Chanel4_DO" := #Signal;   //Канал 4
               5:
                   "Module10Chanel5_DO" := #Signal;   //Канал 5
               6:
                   "Module10Chanel6_DO" := #Signal;   //Канал 6
               7:
                   "Module10Chanel7_DO" := #Signal;   //Канал 7
               8:
                   "Module10Chanel8_DO" := #Signal;   //Канал 8
               9:
                   "Module10Chanel9_DO" := #Signal;   //Канал 9
               10:
                   "Module10Chanel10_DO" := #Signal;   //Канал 10
               11:
                   "Module10Chanel11_DO" := #Signal;   //Канал 11
               12:
                   "Module10Chanel12_DO" := #Signal;   //Канал 12
               13:
                   "Module10Chanel13_DO" := #Signal;   //Канал 13
               14:
                   "Module10Chanel14_DO" := #Signal;   //Канал 14
               15:
                   "Module10Chanel15_DO" := #Signal;   //Канал 15
               16:
                   "Module10Chanel16_DO" := #Signal;   //Канал 16
           END_CASE;
       11:  // Модуль 11
           CASE #N_chanel OF
               1:
                   "Module11Chanel1_DO" := #Signal;   //Канал 1
               2:
                   "Module11Chanel2_DO" := #Signal;   //Канал 2
               3:
                   "Module11Chanel3_DO" := #Signal;   //Канал 3
               4:
                   "Module11Chanel4_DO" := #Signal;   //Канал 4
               5:
                   "Module11Chanel5_DO" := #Signal;   //Канал 5
               6:
                   "Module11Chanel6_DO" := #Signal;   //Канал 6
               7:
                   "Module11Chanel7_DO" := #Signal;   //Канал 7
               8:
                   "Module11Chanel8_DO" := #Signal;   //Канал 8
               9:
                   "Module11Chanel9_DO" := #Signal;   //Канал 9
               10:
                   "Module11Chanel10_DO" := #Signal;   //Канал 10
               11:
                   "Module11Chanel11_DO" := #Signal;   //Канал 11
               12:
                   "Module11Chanel12_DO" := #Signal;   //Канал 12
               13:
                   "Module11Chanel13_DO" := #Signal;   //Канал 13
               14:
                   "Module11Chanel14_DO" := #Signal;   //Канал 14
               15:
                   "Module11Chanel15_DO" := #Signal;   //Канал 15
               16:
                   "Module11Chanel16_DO" := #Signal;   //Канал 16
           END_CASE;
       12:  // Модуль 12
           CASE #N_chanel OF
               1:
                   "Module12Chanel1_DO" := #Signal;   //Канал 1
               2:
                   "Module12Chanel2_DO" := #Signal;   //Канал 2
               3:
                   "Module12Chanel3_DO" := #Signal;   //Канал 3
               4:
                   "Module12Chanel4_DO" := #Signal;   //Канал 4
               5:
                   "Module12Chanel5_DO" := #Signal;   //Канал 5
               6:
                   "Module12Chanel6_DO" := #Signal;   //Канал 6
               7:
                   "Module12Chanel7_DO" := #Signal;   //Канал 7
               8:
                   "Module12Chanel8_DO" := #Signal;   //Канал 8
               9:
                   "Module12Chanel9_DO" := #Signal;   //Канал 9
               10:
                   "Module12Chanel10_DO" := #Signal;   //Канал 10
               11:
                   "Module12Chanel11_DO" := #Signal;   //Канал 11
               12:
                   "Module12Chanel12_DO" := #Signal;   //Канал 12
               13:
                   "Module12Chanel13_DO" := #Signal;   //Канал 13
               14:
                   "Module12Chanel14_DO" := #Signal;   //Канал 14
               15:
                   "Module12Chanel15_DO" := #Signal;   //Канал 15
               16:
                   "Module12Chanel16_DO" := #Signal;   //Канал 16
           END_CASE;
       13:  // Модуль 13
           CASE #N_chanel OF
               1:
                   "Module13Chanel1_DO" := #Signal;   //Канал 1
               2:
                   "Module13Chanel2_DO" := #Signal;   //Канал 2
               3:
                   "Module13Chanel3_DO" := #Signal;   //Канал 3
               4:
                   "Module13Chanel4_DO" := #Signal;   //Канал 4
               5:
                   "Module13Chanel5_DO" := #Signal;   //Канал 5
               6:
                   "Module13Chanel6_DO" := #Signal;   //Канал 6
               7:
                   "Module13Chanel7_DO" := #Signal;   //Канал 7
               8:
                   "Module13Chanel8_DO" := #Signal;   //Канал 8
               9:
                   "Module13Chanel9_DO" := #Signal;   //Канал 9
               10:
                   "Module13Chanel10_DO" := #Signal;   //Канал 10
               11:
                   "Module13Chanel11_DO" := #Signal;   //Канал 11
               12:
                   "Module13Chanel12_DO" := #Signal;   //Канал 12
               13:
                   "Module13Chanel13_DO" := #Signal;   //Канал 13
               14:
                   "Module13Chanel14_DO" := #Signal;   //Канал 14
               15:
                   "Module13Chanel15_DO" := #Signal;   //Канал 15
               16:
                   "Module13Chanel16_DO" := #Signal;   //Канал 16
           END_CASE;
       14:  // Модуль 14
           CASE #N_chanel OF
               1:
                   "Module14Chanel1_DO" := #Signal;   //Канал 1
               2:
                   "Module14Chanel2_DO" := #Signal;   //Канал 2
               3:
                   "Module14Chanel3_DO" := #Signal;   //Канал 3
               4:
                   "Module14Chanel4_DO" := #Signal;   //Канал 4
               5:
                   "Module14Chanel5_DO" := #Signal;   //Канал 5
               6:
                   "Module14Chanel6_DO" := #Signal;   //Канал 6
               7:
                   "Module14Chanel7_DO" := #Signal;   //Канал 7
               8:
                   "Module14Chanel8_DO" := #Signal;   //Канал 8
               9:
                   "Module14Chanel9_DO" := #Signal;   //Канал 9
               10:
                   "Module14Chanel10_DO" := #Signal;   //Канал 10
               11:
                   "Module14Chanel11_DO" := #Signal;   //Канал 11
               12:
                   "Module14Chanel12_DO" := #Signal;   //Канал 12
               13:
                   "Module14Chanel13_DO" := #Signal;   //Канал 13
               14:
                   "Module14Chanel14_DO" := #Signal;   //Канал 14
               15:
                   "Module14Chanel15_DO" := #Signal;   //Канал 15
               16:
                   "Module14Chanel16_DO" := #Signal;   //Канал 16
           END_CASE;
       15:  // Модуль 15
           CASE #N_chanel OF
               1:
                   "Module15Chanel1_DO" := #Signal;   //Канал 1
               2:
                   "Module15Chanel2_DO" := #Signal;   //Канал 2
               3:
                   "Module15Chanel3_DO" := #Signal;   //Канал 3
               4:
                   "Module15Chanel4_DO" := #Signal;   //Канал 4
               5:
                   "Module15Chanel5_DO" := #Signal;   //Канал 5
               6:
                   "Module15Chanel6_DO" := #Signal;   //Канал 6
               7:
                   "Module15Chanel7_DO" := #Signal;   //Канал 7
               8:
                   "Module15Chanel8_DO" := #Signal;   //Канал 8
               9:
                   "Module15Chanel9_DO" := #Signal;   //Канал 9
               10:
                   "Module15Chanel10_DO" := #Signal;   //Канал 10
               11:
                   "Module15Chanel11_DO" := #Signal;   //Канал 11
               12:
                   "Module15Chanel12_DO" := #Signal;   //Канал 12
               13:
                   "Module15Chanel13_DO" := #Signal;   //Канал 13
               14:
                   "Module15Chanel14_DO" := #Signal;   //Канал 14
               15:
                   "Module15Chanel15_DO" := #Signal;   //Канал 15
               16:
                   "Module15Chanel16_DO" := #Signal;   //Канал 16
           END_CASE;
       16:  // Модуль 16
           CASE #N_chanel OF
               1:
                   "Module16Chanel1_DO" := #Signal;   //Канал 1
               2:
                   "Module16Chanel2_DO" := #Signal;   //Канал 2
               3:
                   "Module16Chanel3_DO" := #Signal;   //Канал 3
               4:
                   "Module16Chanel4_DO" := #Signal;   //Канал 4
               5:
                   "Module16Chanel5_DO" := #Signal;   //Канал 5
               6:
                   "Module16Chanel6_DO" := #Signal;   //Канал 6
               7:
                   "Module16Chanel7_DO" := #Signal;   //Канал 7
               8:
                   "Module16Chanel8_DO" := #Signal;   //Канал 8
               9:
                   "Module16Chanel9_DO" := #Signal;   //Канал 9
               10:
                   "Module16Chanel10_DO" := #Signal;   //Канал 10
               11:
                   "Module16Chanel11_DO" := #Signal;   //Канал 11
               12:
                   "Module16Chanel12_DO" := #Signal;   //Канал 12
               13:
                   "Module16Chanel13_DO" := #Signal;   //Канал 13
               14:
                   "Module16Chanel14_DO" := #Signal;   //Канал 14
               15:
                   "Module16Chanel15_DO" := #Signal;   //Канал 15
               16:
                   "Module16Chanel16_DO" := #Signal;   //Канал 16
           END_CASE;
       17:  // Модуль 17
           CASE #N_chanel OF
               1:
                   "Module17Chanel1_DO" := #Signal;   //Канал 1
               2:
                   "Module17Chanel2_DO" := #Signal;   //Канал 2
               3:
                   "Module17Chanel3_DO" := #Signal;   //Канал 3
               4:
                   "Module17Chanel4_DO" := #Signal;   //Канал 4
               5:
                   "Module17Chanel5_DO" := #Signal;   //Канал 5
               6:
                   "Module17Chanel6_DO" := #Signal;   //Канал 6
               7:
                   "Module17Chanel7_DO" := #Signal;   //Канал 7
               8:
                   "Module17Chanel8_DO" := #Signal;   //Канал 8
               9:
                   "Module17Chanel9_DO" := #Signal;   //Канал 9
               10:
                   "Module17Chanel10_DO" := #Signal;   //Канал 10
               11:
                   "Module17Chanel11_DO" := #Signal;   //Канал 11
               12:
                   "Module17Chanel12_DO" := #Signal;   //Канал 12
               13:
                   "Module17Chanel13_DO" := #Signal;   //Канал 13
               14:
                   "Module17Chanel14_DO" := #Signal;   //Канал 14
               15:
                   "Module17Chanel15_DO" := #Signal;   //Канал 15
               16:
                   "Module17Chanel16_DO" := #Signal;   //Канал 16
           END_CASE;
       18:  // Модуль 18
           CASE #N_chanel OF
               1:
                   "Module18Chanel1_DO" := #Signal;   //Канал 1
               2:
                   "Module18Chanel2_DO" := #Signal;   //Канал 2
               3:
                   "Module18Chanel3_DO" := #Signal;   //Канал 3
               4:
                   "Module18Chanel4_DO" := #Signal;   //Канал 4
               5:
                   "Module18Chanel5_DO" := #Signal;   //Канал 5
               6:
                   "Module18Chanel6_DO" := #Signal;   //Канал 6
               7:
                   "Module18Chanel7_DO" := #Signal;   //Канал 7
               8:
                   "Module18Chanel8_DO" := #Signal;   //Канал 8
               9:
                   "Module18Chanel9_DO" := #Signal;   //Канал 9
               10:
                   "Module18Chanel10_DO" := #Signal;   //Канал 10
               11:
                   "Module18Chanel11_DO" := #Signal;   //Канал 11
               12:
                   "Module18Chanel12_DO" := #Signal;   //Канал 12
               13:
                   "Module18Chanel13_DO" := #Signal;   //Канал 13
               14:
                   "Module18Chanel14_DO" := #Signal;   //Канал 14
               15:
                   "Module18Chanel15_DO" := #Signal;   //Канал 15
               16:
                   "Module18Chanel16_DO" := #Signal;   //Канал 16
           END_CASE;
       19:  // Модуль 19
           CASE #N_chanel OF
               1:
                   "Module19Chanel1_DO" := #Signal;   //Канал 1
               2:
                   "Module19Chanel2_DO" := #Signal;   //Канал 2
               3:
                   "Module19Chanel3_DO" := #Signal;   //Канал 3
               4:
                   "Module19Chanel4_DO" := #Signal;   //Канал 4
               5:
                   "Module19Chanel5_DO" := #Signal;   //Канал 5
               6:
                   "Module19Chanel6_DO" := #Signal;   //Канал 6
               7:
                   "Module19Chanel7_DO" := #Signal;   //Канал 7
               8:
                   "Module19Chanel8_DO" := #Signal;   //Канал 8
               9:
                   "Module19Chanel9_DO" := #Signal;   //Канал 9
               10:
                   "Module19Chanel10_DO" := #Signal;   //Канал 10
               11:
                   "Module19Chanel11_DO" := #Signal;   //Канал 11
               12:
                   "Module19Chanel12_DO" := #Signal;   //Канал 12
               13:
                   "Module19Chanel13_DO" := #Signal;   //Канал 13
               14:
                   "Module19Chanel14_DO" := #Signal;   //Канал 14
               15:
                   "Module19Chanel15_DO" := #Signal;   //Канал 15
               16:
                   "Module19Chanel16_DO" := #Signal;   //Канал 16
           END_CASE;
       20:  // Модуль 20
           CASE #N_chanel OF
               1:
                   "Module20Chanel1_DO" := #Signal;   //Канал 1
               2:
                   "Module20Chanel2_DO" := #Signal;   //Канал 2
               3:
                   "Module20Chanel3_DO" := #Signal;   //Канал 3
               4:
                   "Module20Chanel4_DO" := #Signal;   //Канал 4
               5:
                   "Module20Chanel5_DO" := #Signal;   //Канал 5
               6:
                   "Module20Chanel6_DO" := #Signal;   //Канал 6
               7:
                   "Module20Chanel7_DO" := #Signal;   //Канал 7
               8:
                   "Module20Chanel8_DO" := #Signal;   //Канал 8
               9:
                   "Module20Chanel9_DO" := #Signal;   //Канал 9
               10:
                   "Module20Chanel10_DO" := #Signal;   //Канал 10
               11:
                   "Module20Chanel11_DO" := #Signal;   //Канал 11
               12:
                   "Module20Chanel12_DO" := #Signal;   //Канал 12
               13:
                   "Module20Chanel13_DO" := #Signal;   //Канал 13
               14:
                   "Module20Chanel14_DO" := #Signal;   //Канал 14
               15:
                   "Module20Chanel15_DO" := #Signal;   //Канал 15
               16:
                   "Module20Chanel16_DO" := #Signal;   //Канал 16
           END_CASE;
       21:  // Модуль 21
           CASE #N_chanel OF
               1:
                   "Module21Chanel1_DO" := #Signal;   //Канал 1
               2:
                   "Module21Chanel2_DO" := #Signal;   //Канал 2
               3:
                   "Module21Chanel3_DO" := #Signal;   //Канал 3
               4:
                   "Module21Chanel4_DO" := #Signal;   //Канал 4
               5:
                   "Module21Chanel5_DO" := #Signal;   //Канал 5
               6:
                   "Module21Chanel6_DO" := #Signal;   //Канал 6
               7:
                   "Module21Chanel7_DO" := #Signal;   //Канал 7
               8:
                   "Module21Chanel8_DO" := #Signal;   //Канал 8
               9:
                   "Module21Chanel9_DO" := #Signal;   //Канал 9
               10:
                   "Module21Chanel10_DO" := #Signal;   //Канал 10
               11:
                   "Module21Chanel11_DO" := #Signal;   //Канал 11
               12:
                   "Module21Chanel12_DO" := #Signal;   //Канал 12
               13:
                   "Module21Chanel13_DO" := #Signal;   //Канал 13
               14:
                   "Module21Chanel14_DO" := #Signal;   //Канал 14
               15:
                   "Module21Chanel15_DO" := #Signal;   //Канал 15
               16:
                   "Module21Chanel16_DO" := #Signal;   //Канал 16
           END_CASE;
       22:  // Модуль 22
           CASE #N_chanel OF
               1:
                   "Module22Chanel1_DO" := #Signal;   //Канал 1
               2:
                   "Module22Chanel2_DO" := #Signal;   //Канал 2
               3:
                   "Module22Chanel3_DO" := #Signal;   //Канал 3
               4:
                   "Module22Chanel4_DO" := #Signal;   //Канал 4
               5:
                   "Module22Chanel5_DO" := #Signal;   //Канал 5
               6:
                   "Module22Chanel6_DO" := #Signal;   //Канал 6
               7:
                   "Module22Chanel7_DO" := #Signal;   //Канал 7
               8:
                   "Module22Chanel8_DO" := #Signal;   //Канал 8
               9:
                   "Module22Chanel9_DO" := #Signal;   //Канал 9
               10:
                   "Module22Chanel10_DO" := #Signal;   //Канал 10
               11:
                   "Module22Chanel11_DO" := #Signal;   //Канал 11
               12:
                   "Module22Chanel12_DO" := #Signal;   //Канал 12
               13:
                   "Module22Chanel13_DO" := #Signal;   //Канал 13
               14:
                   "Module22Chanel14_DO" := #Signal;   //Канал 14
               15:
                   "Module22Chanel15_DO" := #Signal;   //Канал 15
               16:
                   "Module22Chanel16_DO" := #Signal;   //Канал 16
           END_CASE;
       23:  // Модуль 23
           CASE #N_chanel OF
               1:
                   "Module23Chanel1_DO" := #Signal;   //Канал 1
               2:
                   "Module23Chanel2_DO" := #Signal;   //Канал 2
               3:
                   "Module23Chanel3_DO" := #Signal;   //Канал 3
               4:
                   "Module23Chanel4_DO" := #Signal;   //Канал 4
               5:
                   "Module23Chanel5_DO" := #Signal;   //Канал 5
               6:
                   "Module23Chanel6_DO" := #Signal;   //Канал 6
               7:
                   "Module23Chanel7_DO" := #Signal;   //Канал 7
               8:
                   "Module23Chanel8_DO" := #Signal;   //Канал 8
               9:
                   "Module23Chanel9_DO" := #Signal;   //Канал 9
               10:
                   "Module23Chanel10_DO" := #Signal;   //Канал 10
               11:
                   "Module23Chanel11_DO" := #Signal;   //Канал 11
               12:
                   "Module23Chanel12_DO" := #Signal;   //Канал 12
               13:
                   "Module23Chanel13_DO" := #Signal;   //Канал 13
               14:
                   "Module23Chanel14_DO" := #Signal;   //Канал 14
               15:
                   "Module23Chanel15_DO" := #Signal;   //Канал 15
               16:
                   "Module23Chanel16_DO" := #Signal;   //Канал 16
           END_CASE;
       24:  // Модуль 24
           CASE #N_chanel OF
               1:
                   "Module24Chanel1_DO" := #Signal;   //Канал 1
               2:
                   "Module24Chanel2_DO" := #Signal;   //Канал 2
               3:
                   "Module24Chanel3_DO" := #Signal;   //Канал 3
               4:
                   "Module24Chanel4_DO" := #Signal;   //Канал 4
               5:
                   "Module24Chanel5_DO" := #Signal;   //Канал 5
               6:
                   "Module24Chanel6_DO" := #Signal;   //Канал 6
               7:
                   "Module24Chanel7_DO" := #Signal;   //Канал 7
               8:
                   "Module24Chanel8_DO" := #Signal;   //Канал 8
               9:
                   "Module24Chanel9_DO" := #Signal;   //Канал 9
               10:
                   "Module24Chanel10_DO" := #Signal;   //Канал 10
               11:
                   "Module24Chanel11_DO" := #Signal;   //Канал 11
               12:
                   "Module24Chanel12_DO" := #Signal;   //Канал 12
               13:
                   "Module24Chanel13_DO" := #Signal;   //Канал 13
               14:
                   "Module24Chanel14_DO" := #Signal;   //Канал 14
               15:
                   "Module24Chanel15_DO" := #Signal;   //Канал 15
               16:
                   "Module24Chanel16_DO" := #Signal;   //Канал 16
           END_CASE;
       25:  // Модуль 25
           CASE #N_chanel OF
               1:
                   "Module25Chanel1_DO" := #Signal;   //Канал 1
               2:
                   "Module25Chanel2_DO" := #Signal;   //Канал 2
               3:
                   "Module25Chanel3_DO" := #Signal;   //Канал 3
               4:
                   "Module25Chanel4_DO" := #Signal;   //Канал 4
               5:
                   "Module25Chanel5_DO" := #Signal;   //Канал 5
               6:
                   "Module25Chanel6_DO" := #Signal;   //Канал 6
               7:
                   "Module25Chanel7_DO" := #Signal;   //Канал 7
               8:
                   "Module25Chanel8_DO" := #Signal;   //Канал 8
               9:
                   "Module25Chanel9_DO" := #Signal;   //Канал 9
               10:
                   "Module25Chanel10_DO" := #Signal;   //Канал 10
               11:
                   "Module25Chanel11_DO" := #Signal;   //Канал 11
               12:
                   "Module25Chanel12_DO" := #Signal;   //Канал 12
               13:
                   "Module25Chanel13_DO" := #Signal;   //Канал 13
               14:
                   "Module25Chanel14_DO" := #Signal;   //Канал 14
               15:
                   "Module25Chanel15_DO" := #Signal;   //Канал 15
               16:
                   "Module25Chanel16_DO" := #Signal;   //Канал 16
           END_CASE;
   END_CASE;
END_FUNCTION

FUNCTION "write_4_20" : Void   // FC7, SCL
{ S7_Optimized_Access := 'TRUE' }
AUTHOR : Dmitriy_Petrov
VERSION : 0.1
// Функция записи сигнала 4-20mA
   VAR_INPUT
      Value : Real;   // Значение в физической величине
      LL_control_signal : Real;   // Нижний предел управляющего воздействия в физической величине
      HL_control_signal : Real;   // Верхний предел управляющего воздействия в физической величине
   END_VAR
   VAR_IN_OUT
      N_module : USInt;   // № модуля (начиная с 1)
      N_chanel : USInt;   // № канала (начиная с 1)
      ADC : Int;   // Текущий код АЦП
   END_VAR
   VAR_TEMP
      K : Real;   // Коэффициент К
      "B" : Real;   // Коэффициент B
   END_VAR
   VAR CONSTANT
      LL_ADC : Int;   // Нижний предел АЦП
      HL_ADC : Int := 27648;   // Верхний предел АЦП
   END_VAR
BEGIN
   (*проверка правильности введеного значения № Модуля*)
   IF #N_module < 1 OR #N_module > 25 THEN
       #N_module := 0;
   END_IF;

   (*проверка правильности введеного значения № Канала*)
   IF #N_module = 0 THEN
       #N_chanel := 0;
   ELSE
       IF #N_chanel < 1 OR #N_chanel > 4 THEN
           #N_chanel := 0;
       END_IF;
   END_IF;

   (*Вычисление кода ЦАП*)
   #K := (#HL_ADC - #LL_ADC) / (#HL_control_signal - #LL_control_signal);
   #"B" := #LL_ADC - (#K * #LL_control_signal);
   #ADC := REAL_TO_INT((#K * #Value) + #"B");

   (*запись кода ЦАП в выбранной канал*)
   CASE #N_module OF
       1:  // Модуль 1
           CASE #N_chanel OF
               1:
                   "Module01Chanel1_AO" := #ADC;   //Канал 1
               2:
                   "Module01Chanel2_AO" := #ADC;   //Канал 2
               3:
                   "Module01Chanel3_AO" := #ADC;   //Канал 3
               4:
                   "Module01Chanel4_AO" := #ADC;   //Канал 4
           END_CASE;
       2:  // Модуль 2
           CASE #N_chanel OF
               1:
                   "Module02Chanel1_AO" := #ADC;   //Канал 1
               2:
                   "Module02Chanel2_AO" := #ADC;   //Канал 2
               3:
                   "Module02Chanel3_AO" := #ADC;   //Канал 3
               4:
                   "Module02Chanel4_AO" := #ADC;   //Канал 4
           END_CASE;
       3:  // Модуль 3
           CASE #N_chanel OF
               1:
                   "Module03Chanel1_AO" := #ADC;   //Канал 1
               2:
                   "Module03Chanel2_AO" := #ADC;   //Канал 2
               3:
                   "Module03Chanel3_AO" := #ADC;   //Канал 3
               4:
                   "Module03Chanel4_AO" := #ADC;   //Канал 4
           END_CASE;
       4:  // Модуль 4
           CASE #N_chanel OF
               1:
                   "Module04Chanel1_AO" := #ADC;   //Канал 1
               2:
                   "Module04Chanel2_AO" := #ADC;   //Канал 2
               3:
                   "Module04Chanel3_AO" := #ADC;   //Канал 3
               4:
                   "Module04Chanel4_AO" := #ADC;   //Канал 4
           END_CASE;
       5:  // Модуль 5
           CASE #N_chanel OF
               1:
                   "Module05Chanel1_AO" := #ADC;   //Канал 1
               2:
                   "Module05Chanel2_AO" := #ADC;   //Канал 2
               3:
                   "Module05Chanel3_AO" := #ADC;   //Канал 3
               4:
                   "Module05Chanel4_AO" := #ADC;   //Канал 4
           END_CASE;
       6:  // Модуль 6
           CASE #N_chanel OF
               1:
                   "Module06Chanel1_AO" := #ADC;   //Канал 1
               2:
                   "Module06Chanel2_AO" := #ADC;   //Канал 2
               3:
                   "Module06Chanel3_AO" := #ADC;   //Канал 3
               4:
                   "Module06Chanel4_AO" := #ADC;   //Канал 4
           END_CASE;
       7:  // Модуль 7
           CASE #N_chanel OF
               1:
                   "Module07Chanel1_AO" := #ADC;   //Канал 1
               2:
                   "Module07Chanel2_AO" := #ADC;   //Канал 2
               3:
                   "Module07Chanel3_AO" := #ADC;   //Канал 3
               4:
                   "Module07Chanel4_AO" := #ADC;   //Канал 4
           END_CASE;
       8:  // Модуль 8
           CASE #N_chanel OF
               1:
                   "Module08Chanel1_AO" := #ADC;   //Канал 1
               2:
                   "Module08Chanel2_AO" := #ADC;   //Канал 2
               3:
                   "Module08Chanel3_AO" := #ADC;   //Канал 3
               4:
                   "Module08Chanel4_AO" := #ADC;   //Канал 4
           END_CASE;
       9:  // Модуль 9
           CASE #N_chanel OF
               1:
                   "Module09Chanel1_AO" := #ADC;   //Канал 1
               2:
                   "Module09Chanel2_AO" := #ADC;   //Канал 2
               3:
                   "Module09Chanel3_AO" := #ADC;   //Канал 3
               4:
                   "Module09Chanel4_AO" := #ADC;   //Канал 4
           END_CASE;
       10:  // Модуль 10
           CASE #N_chanel OF
               1:
                   "Module10Chanel1_AO" := #ADC;   //Канал 1
               2:
                   "Module10Chanel2_AO" := #ADC;   //Канал 2
               3:
                   "Module10Chanel3_AO" := #ADC;   //Канал 3
               4:
                   "Module10Chanel4_AO" := #ADC;   //Канал 4
           END_CASE;
       11:  // Модуль 11
           CASE #N_chanel OF
               1:
                   "Module11Chanel1_AO" := #ADC;   //Канал 1
               2:
                   "Module11Chanel2_AO" := #ADC;   //Канал 2
               3:
                   "Module11Chanel3_AO" := #ADC;   //Канал 3
               4:
                   "Module11Chanel4_AO" := #ADC;   //Канал 4
           END_CASE;
       12:  // Модуль 12
           CASE #N_chanel OF
               1:
                   "Module12Chanel1_AO" := #ADC;   //Канал 1
               2:
                   "Module12Chanel2_AO" := #ADC;   //Канал 2
               3:
                   "Module12Chanel3_AO" := #ADC;   //Канал 3
               4:
                   "Module12Chanel4_AO" := #ADC;   //Канал 4
           END_CASE;
       13:  // Модуль 13
           CASE #N_chanel OF
               1:
                   "Module13Chanel1_AO" := #ADC;   //Канал 1
               2:
                   "Module13Chanel2_AO" := #ADC;   //Канал 2
               3:
                   "Module13Chanel3_AO" := #ADC;   //Канал 3
               4:
                   "Module13Chanel4_AO" := #ADC;   //Канал 4
           END_CASE;
       14:  // Модуль 14
           CASE #N_chanel OF
               1:
                   "Module14Chanel1_AO" := #ADC;   //Канал 1
               2:
                   "Module14Chanel2_AO" := #ADC;   //Канал 2
               3:
                   "Module14Chanel3_AO" := #ADC;   //Канал 3
               4:
                   "Module14Chanel4_AO" := #ADC;   //Канал 4
           END_CASE;
       15:  // Модуль 15
           CASE #N_chanel OF
               1:
                   "Module15Chanel1_AO" := #ADC;   //Канал 1
               2:
                   "Module15Chanel2_AO" := #ADC;   //Канал 2
               3:
                   "Module15Chanel3_AO" := #ADC;   //Канал 3
               4:
                   "Module15Chanel4_AO" := #ADC;   //Канал 4
           END_CASE;
       16:  // Модуль 16
           CASE #N_chanel OF
               1:
                   "Module16Chanel1_AO" := #ADC;   //Канал 1
               2:
                   "Module16Chanel2_AO" := #ADC;   //Канал 2
               3:
                   "Module16Chanel3_AO" := #ADC;   //Канал 3
               4:
                   "Module16Chanel4_AO" := #ADC;   //Канал 4
           END_CASE;
       17:  // Модуль 17
           CASE #N_chanel OF
               1:
                   "Module17Chanel1_AO" := #ADC;   //Канал 1
               2:
                   "Module17Chanel2_AO" := #ADC;   //Канал 2
               3:
                   "Module17Chanel3_AO" := #ADC;   //Канал 3
               4:
                   "Module17Chanel4_AO" := #ADC;   //Канал 4
           END_CASE;
       18:  // Модуль 18
           CASE #N_chanel OF
               1:
                   "Module18Chanel1_AO" := #ADC;   //Канал 1
               2:
                   "Module18Chanel2_AO" := #ADC;   //Канал 2
               3:
                   "Module18Chanel3_AO" := #ADC;   //Канал 3
               4:
                   "Module18Chanel4_AO" := #ADC;   //Канал 4
           END_CASE;
       19:  // Модуль 19
           CASE #N_chanel OF
               1:
                   "Module19Chanel1_AO" := #ADC;   //Канал 1
               2:
                   "Module19Chanel2_AO" := #ADC;   //Канал 2
               3:
                   "Module19Chanel3_AO" := #ADC;   //Канал 3
               4:
                   "Module19Chanel4_AO" := #ADC;   //Канал 4
           END_CASE;
       20:  // Модуль 20
           CASE #N_chanel OF
               1:
                   "Module20Chanel1_AO" := #ADC;   //Канал 1
               2:
                   "Module20Chanel2_AO" := #ADC;   //Канал 2
               3:
                   "Module20Chanel3_AO" := #ADC;   //Канал 3
               4:
                   "Module20Chanel4_AO" := #ADC;   //Канал 4
           END_CASE;
       21:  // Модуль 21
           CASE #N_chanel OF
               1:
                   "Module21Chanel1_AO" := #ADC;   //Канал 1
               2:
                   "Module21Chanel2_AO" := #ADC;   //Канал 2
               3:
                   "Module21Chanel3_AO" := #ADC;   //Канал 3
               4:
                   "Module21Chanel4_AO" := #ADC;   //Канал 4
           END_CASE;
       22:  // Модуль 22
           CASE #N_chanel OF
               1:
                   "Module22Chanel1_AO" := #ADC;   //Канал 1
               2:
                   "Module22Chanel2_AO" := #ADC;   //Канал 2
               3:
                   "Module22Chanel3_AO" := #ADC;   //Канал 3
               4:
                   "Module22Chanel4_AO" := #ADC;   //Канал 4
           END_CASE;
       23:  // Модуль 23
           CASE #N_chanel OF
               1:
                   "Module23Chanel1_AO" := #ADC;   //Канал 1
               2:
                   "Module23Chanel2_AO" := #ADC;   //Канал 2
               3:
                   "Module23Chanel3_AO" := #ADC;   //Канал 3
               4:
                   "Module23Chanel4_AO" := #ADC;   //Канал 4
           END_CASE;
       24:  // Модуль 24
           CASE #N_chanel OF
               1:
                   "Module24Chanel1_AO" := #ADC;   //Канал 1
               2:
                   "Module24Chanel2_AO" := #ADC;   //Канал 2
               3:
                   "Module24Chanel3_AO" := #ADC;   //Канал 3
               4:
                   "Module24Chanel4_AO" := #ADC;   //Канал 4
           END_CASE;
       25:  // Модуль 25
           CASE #N_chanel OF
               1:
                   "Module25Chanel1_AO" := #ADC;   //Канал 1
               2:
                   "Module25Chanel2_AO" := #ADC;   //Канал 2
               3:
                   "Module25Chanel3_AO" := #ADC;   //Канал 3
               4:
                   "Module25Chanel4_AO" := #ADC;   //Канал 4
           END_CASE;
   END_CASE;
END_FUNCTION

FUNCTION "HMI_and_SCADA" : Void   // FC8, SCL
{ S7_Optimized_Access := 'TRUE' }
VERSION : 0.1
BEGIN
   //кнопка ВЕНТИЛЯЦИЯ на панели оператора
   "R_TRIG_DB"(CLK := "HMI".Btn_Ventilation_HMI,
               Q => "FRONT".Btn_Ventilation_HMI);
   IF "FRONT".Btn_Ventilation_HMI THEN
       "HMI".Btn_Ventilation_HMI := FALSE;
   END_IF;
   //кнопка ВЕНТИЛЯЦИЯ на SCADA
   "R_TRIG_DB_1"(CLK := "HMI".Btn_Ventilation_SCADA,
                 Q => "FRONT".Btn_Ventilation_SCADA);
   IF "FRONT".Btn_Ventilation_SCADA THEN
       "HMI".Btn_Ventilation_SCADA := FALSE;
   END_IF;
   //кнопка РОЗЖИГ на панели оператора
   "R_TRIG_DB_2"(CLK := "HMI".Btn_Ignition_HMI,
                 Q => "FRONT".Btn_Ignition_HMI);
   IF "FRONT".Btn_Ignition_HMI THEN
       "HMI".Btn_Ignition_HMI := FALSE;
   END_IF;
   //кнопка РОЗЖИГ на SCADA
   "R_TRIG_DB_3"(CLK := "HMI".Btn_Ignition_SCADA,
                 Q => "FRONT".Btn_Ignition_SCADA);
   IF "FRONT".Btn_Ignition_SCADA THEN
       "HMI".Btn_Ignition_SCADA := FALSE;
   END_IF;
   //кнопка НОРМАЛЬНЫЙ ОСТАНОВ на панели оператора
   "R_TRIG_DB_4"(CLK := "HMI".Btn_normal_stop_HMI,
                 Q => "FRONT".Btn_Normal_stop_HMI);
   IF "FRONT".Btn_Normal_stop_HMI THEN
       "HMI".Btn_normal_stop_HMI := FALSE;
   END_IF;
   //кнопка НОРМАЛЬНЫЙ ОСТАНОВ на SCADA
   "R_TRIG_DB_5"(CLK := "HMI".Btn_normal_stop_SCADA,
                 Q => "FRONT".Btn_Normal_stop_SCADA);
   IF "FRONT".Btn_Normal_stop_SCADA THEN
       "HMI".Btn_normal_stop_SCADA := FALSE;
   END_IF;
   //кнопка АВАРИЙНЫЙ ОСТАНОВ на панели оператора
   "R_TRIG_DB_6"(CLK := "HMI".Btn_alarm_stop_HMI,
                 Q => "FRONT".Btn_Alarm_stop_HMI);
   IF "FRONT".Btn_Alarm_stop_HMI THEN
       "HMI".Btn_alarm_stop_HMI := FALSE;
   END_IF;
   //кнопка АВАРИЙНЫЙ ОСТАНОВ на SCADA
   "R_TRIG_DB_7"(CLK := "HMI".Btn_alarm_stop_SCADA,
                 Q => "FRONT".Btn_Alarm_stop_SCADA);
   IF "FRONT".Btn_Alarm_stop_SCADA THEN
       "HMI".Btn_alarm_stop_SCADA := FALSE;
   END_IF;
   //кнопка ТЕСТОВАЯ ОПРЕССОВКА на панели оператора
   "R_TRIG_DB_8"(CLK := "HMI".Btn_test_press_HMI,
                 Q => "FRONT".Btn_test_press_HMI);
   IF "FRONT".Btn_test_press_HMI THEN
       "HMI".Btn_test_press_HMI := FALSE;
   END_IF;
   //кнопка ТЕСТОВЫЙ РОЗЖИГ на панели оператора
   "R_TRIG_DB_9"(CLK := "HMI".Btn_test_ignition_HMI,
                 Q => "FRONT".Btn_test_ignition_HMI);
   IF "FRONT".Btn_test_ignition_HMI THEN
       "HMI".Btn_test_ignition_HMI := FALSE;
   END_IF;

   //кнопка РУЧНОЙ РОЗЖИГ на панели оператора
   (* "R_TRIG_DB_10"(CLK:="HMI".Btn_manual_ignition_HMI,
                  Q =>"FRONT_Btn_manual_ignition_HMI");
   IF "FRONT_Btn_manual_ignition_HMI" THEN
       "HMI".Btn_manual_ignition_HMI := FALSE;
   END_IF; *)
   IF NOT ("Technology".Regim = 3 AND "Technology".Regim_ventilation_step = 25) AND NOT ("Technology".Regim = 5 AND "Technology".Regim_ignition_step = 19) THEN
       "HMI".Btn_manual_ignition_HMI := FALSE;
   END_IF;

   //кнопка СБРОС ЗВУКА на панели оператора
   "R_TRIG_DB_28"(CLK := "HMI".Btn_reset_sound_HMI,
                  Q => "FRONT".Btn_reset_sound_HMI);
   IF "FRONT".Btn_reset_sound_HMI THEN
       "HMI".Btn_reset_sound_HMI := FALSE;
   END_IF;

   (*Текущая уставка регулятора давления воздуха*)
   IF "DV_invertor_mode".Value THEN
       "HMI".Current_SP_P_air := "Control_DV".SP_PID;
   END_IF;
   IF "DV_powergrid_mode".Value THEN
       "HMI".Current_SP_P_air := "Control_NAV".SP_PID;
   END_IF;
   (*Текущая уставка регулятора разряжения*)
   IF "DS_invertor_mode".Value THEN
       "HMI".Current_SP_dP_furnance := "Control_DS".SP_PID;
   END_IF;
   IF "DS_powergrid_mode".Value THEN
       "HMI".Current_SP_dP_furnance := "Control_NAD".SP_PID;
   END_IF;

   (*Определение текущего подрежима*)
   CASE "Technology".Regim OF
       1:  //откл
           "HMI".INDICATION_TIME_1 := 255;
           "HMI".INDICATION_TIME_2 := 255;
           CASE "Technology".Regim_off_step OF
               0:
                   "Technology".Substage := 1; //перевод ИМ в дистанционный режим

               1:
                   "HMI".INDICATION_TIME_1 := 255;
                   "HMI".INDICATION_TIME_2 := 255;

                   IF "Message".VENTILATION_not_initial_state_air THEN
                       "Technology".Substage := 11; //НАД, НАВ не закрылись или не откл ДВ
                   ELSE
                       IF "Message".VENTILATION_NAV_not_close THEN
                           "Technology".Substage := 13; //НАВ не закрылся
                       ELSE
                           "Technology".Substage := 2; //ожидание нажатия кн.Вентиляция
                           //"Technology".Substage := 168; //ожидание дальнейших действий. Нажмите кн.Вентиляция или кн.Плановый останов
                       END_IF;
                   END_IF;

               2:
                   "HMI".INDICATION_TIME_1 := 255;
                   "HMI".INDICATION_TIME_2 := 255;
                   "Technology".Substage := 4; //перевод газовых клапанов в исходное положение

               3:
                   "HMI".INDICATION_TIME_1 := 255;
                   "HMI".INDICATION_TIME_2 := 255;
                   "Technology".Substage := 169; //отключение ДВ
               4:
                   "HMI".INDICATION_TIME_1 := 255;
                   "HMI".INDICATION_TIME_2 := 255;
                   "Technology".Substage := 170; //отключение ДС             
               ELSE
                   "Technology".Substage := 0; //неизвестно
           END_CASE;
       3:  //вентиляция
           CASE "Technology".Regim_ventilation_step OF
               0:
                   "HMI".INDICATION_TIME_1 := 255;
                   "HMI".INDICATION_TIME_2 := 255;
                   "Technology".Substage := 3; //проверка положения газовых клапанов (не используется)
               1:
                   "HMI".INDICATION_TIME_1 := 255;
                   "HMI".INDICATION_TIME_2 := 255;
                   IF NOT "Message".VENTILATION_not_initial_state_gas THEN
                       "Technology".Substage := 4; //перевод газовых клапанов в исходное положение
                   ELSE
                       "Technology".Substage := 5; //газовые клапана не перевелись в исходное положение
                   END_IF;
               2:
                   "HMI".INDICATION_TIME_1 := 255;
                   "HMI".INDICATION_TIME_2 := 255;
                   IF NOT "Message".VENTILATION_DS_need_dist_mode THEN
                       "Technology".Substage := 6; //проверка нахождения ШУД ДС в дистанционном режиме
                   ELSE
                       "Technology".Substage := 7; //необходимо перевести ШУД ДС в дистанционный режим
                   END_IF;
               3:
                   "HMI".INDICATION_TIME_1 := 255;
                   "HMI".INDICATION_TIME_2 := 255;
                   IF NOT "Message".VENTILATION_DV_need_dist_mode THEN
                       "Technology".Substage := 8; //проверка нахождения ШУД ДВ в дистанционном режиме
                   ELSE
                       "Technology".Substage := 9; //необходимо перевести ШУД ДВ в дистанционный режим
                   END_IF;
               4:
                   IF NOT "Message".VENTILATION_BRU_NAD_need_avto_mode THEN
                       "Technology".Substage := 171;   //проверка нахождения БРУ НАД в автоматическом режиме
                   ELSE
                       "Technology".Substage := 172;   //необходимо перевести БРУ НАД в автоматический режим
                   END_IF;
               5:
                   IF NOT "Message".VENTILATION_BRU_NAV_need_avto_mode THEN
                       "Technology".Substage := 173;   //проверка нахождения БРУ НАВ в автоматическом режиме
                   ELSE
                       "Technology".Substage := 174;   //необходимо перевести БРУ НАВ в автоматический режим
                   END_IF;
               6:
                   "HMI".INDICATION_TIME_1 := 255;
                   "HMI".INDICATION_TIME_2 := 255;
                   IF NOT "Message".VENTILATION_not_initial_state_air THEN
                       "Technology".Substage := 10; //закрытие НАД, НАВ, откл ДВ
                   ELSE
                       "Technology".Substage := 11; //НАД, НАВ не закрылись или не откл ДВ
                   END_IF;
               7:
                   "HMI".INDICATION_TIME_1 := 255;
                   "HMI".INDICATION_TIME_2 := 255;
                   IF NOT "Message".VENTILATION_NAV_not_close THEN
                       "Technology".Substage := 12; //закрытие НАВ
                   ELSE
                       "Technology".Substage := 13; //НАВ не закрылся
                   END_IF;
               8:
                   "HMI".INDICATION_TIME_1 := 255;
                   "HMI".INDICATION_TIME_2 := 255;
                   "Technology".Substage := 14; //проверка состояния ДС
               9:
                   "HMI".INDICATION_TIME_1 := 255;
                   "HMI".INDICATION_TIME_2 := 255;
                   IF NOT "Message".VENTILATION_DS_not_on THEN
                       "Technology".Substage := 15; //пуск ДС
                   ELSE
                       "Technology".Substage := 16; //ДС не включился
                   END_IF;
               10:
                   "HMI".INDICATION_TIME_1 := 255;
                   "HMI".INDICATION_TIME_2 := 255;
                   "Technology".Substage := 15; //пуск ДС
               11:
                   "HMI".INDICATION_TIME_1 := 255;
                   "HMI".INDICATION_TIME_2 := 255;
                   "Technology".Substage := 17; //проверка состояния ДВ
               12:
                   "HMI".INDICATION_TIME_1 := 255;
                   "HMI".INDICATION_TIME_2 := 255;
                   IF NOT "Message".VENTILATION_DV_not_on THEN
                       "Technology".Substage := 18; //пуск ДВ
                   ELSE
                       "Technology".Substage := 19; //ДВ не включился
                   END_IF;
               13:
                   "HMI".INDICATION_TIME_1 := 255;
                   "HMI".INDICATION_TIME_2 := 255;
                   "Technology".Substage := 18; //пуск ДВ
               14:
                   "HMI".INDICATION_TIME_1 := 255;
                   "HMI".INDICATION_TIME_2 := 255;
                   IF NOT "Message".VENTILATION_NAD_not_open_manual THEN
                       "Technology".Substage := 20; //открытие НАД
                   ELSE
                       "Technology".Substage := 21; //БРУ НАД в местром режиме и НАД не открыт
                   END_IF;
                   (* IF NOT "Message".VENTILATION_NAD_not_open THEN
                       "Technology".Substage := 20; //открытие НАД
                   ELSE
                       "Technology".Substage := 21; //НАД не открылся
                   END_IF; *)
               15:
                   "HMI".INDICATION_TIME_1 := 255;
                   "HMI".INDICATION_TIME_2 := 255;
                   "Technology".Substage := 20; //открытие НАД
               16:
                   "HMI".INDICATION_TIME_1 := 255;
                   "HMI".INDICATION_TIME_2 := 255;

                   IF NOT "Message".VENTILATION_NAV_not_open_manual THEN
                       IF NOT "Message".VENTILATION_NAV_or_NAD_not_open THEN
                           "Technology".Substage := 22; //открытие НАВ и НАД
                       ELSE
                           "Technology".Substage := 23; //НАВ или НАД не открылись
                       END_IF;
                   ELSE
                       "Technology".Substage := 33; //БРУ НАВ в местром режиме и НАВ не открыт
                   END_IF;
               17:
                   "HMI".INDICATION_TIME_1 := 255;
                   "HMI".INDICATION_TIME_2 := 255;
                   "Technology".Substage := 22; //открытие НАВ и НАД
               18:
                   "HMI".INDICATION_TIME_1 := 255;
                   "HMI".INDICATION_TIME_2 := 255;
                   "Technology".Substage := 24; //Включаем ПИД ДС на вентиляционные параметры
               19:
                   "HMI".INDICATION_TIME_1 := 255;
                   "HMI".INDICATION_TIME_2 := 255;
                   "Technology".Substage := 24; //Включаем ПИД ДС на вентиляционные параметры
               20:
                   "HMI".INDICATION_TIME_1 := 255;
                   "HMI".INDICATION_TIME_2 := 255;
                   "Technology".Substage := 25; //Включаем ПИД ДВ на вентиляционные параметры
               21:
                   "HMI".INDICATION_TIME_1 := 255;
                   "HMI".INDICATION_TIME_2 := 255;
                   "Technology".Substage := 25; //Включаем ПИД ДВ на вентиляционные параметры
               22:
                   "HMI".INDICATION_TIME_1 := 255;
                   "HMI".INDICATION_TIME_2 := 255;
                   "Technology".Substage := 26; //Проверка достижения вентиляционных параметров
               23:
                   "HMI".TIME_converter_IN := "Timer_VENTILATION_DB".PT - "Timer_VENTILATION_DB".ET;
                   "HMI".INDICATION_TIME_1 := INT_TO_USINT("HMI".TIME_converter_minute);
                   "HMI".INDICATION_TIME_2 := INT_TO_USINT("HMI".TIME_converter_second);

                   IF "Message".VENTILATION_run THEN
                       "Technology".Substage := 27; //вентиляция топки
                   ELSE
                       "Technology".Substage := 28; //параметры вентиляции не в норме
                   END_IF;
               24:
                   "HMI".INDICATION_TIME_1 := 255;
                   "HMI".INDICATION_TIME_2 := 255;
                   "Technology".Substage := 29; //вентиляция прервана. Устраните неисправность. Для повторного проведения нажмите кн.Вентиляция. Для останова нажмите кн.Плановый останов
               25:
                   "HMI".INDICATION_TIME_1 := 255;
                   "HMI".INDICATION_TIME_2 := 255;
                   IF NOT "Message".VENTILATION_Check_param THEN
                       IF NOT "Message".TEST_PRESS_ok THEN
                           "Technology".Substage := 30; //вентиляция проведена. Ожидание дальнейших действий
                       ELSE
                           "Technology".Substage := 31; //тестовая опрессовка успешно проведена
                       END_IF;
                   ELSE
                       "Technology".Substage := 32; //переход невозможен. Проверьте параметры вентиляции
                   END_IF;
               ELSE
                   "HMI".INDICATION_TIME_1 := 255;
                   "HMI".INDICATION_TIME_2 := 255;
                   "Technology".Substage := 0; //неизвестно
           END_CASE;
       4:  //опрессовка
           "HMI".INDICATION_TIME_1 := 255;
           "HMI".INDICATION_TIME_2 := 255;
           CASE "Technology".Regim_press_step OF
               0:
                   "Technology".Substage := 40; //открытие ЗДСВ
               1:
                   "Technology".Substage := 41; //перевод регулятора разрежения на розжиговые параметры
               2:
                   "Technology".Substage := 42; //перевод регулятора разрежения на розжиговые параметры
               3:
                   "Technology".Substage := 43; //перевод регулятора давления воздуха на розжиговые параметры
               4:
                   "Technology".Substage := 44; //перевод регулятора давления воздуха на розжиговые параметры
               5:
                   "Technology".Substage := 45; //проверка достижения розжиговых параметров
               6:
                   IF NOT "Message".PRESS_not_initial_state_gas THEN
                       "Technology".Substage := 46; //перевод клапанов по газу в исходное состояние
                   ELSE
                       "Technology".Substage := 47; //клапана по газу не переведены в исходное состояние
                   END_IF;
               7:
                   IF NOT "Message".PRESS_ZRG_not_close THEN
                       "Technology".Substage := 48; //закрываем ЗРГ
                   ELSE
                       "Technology".Substage := 49; //ЗРГ не закрылся
                   END_IF;
               8:
                   IF NOT "Message".PRESS_ZDG_not_open THEN
                       "Technology".Substage := 50; //открываем ЗДГ
                   ELSE
                       "Technology".Substage := 51; //ЗДГ не открылся
                   END_IF;
               9:
                   "Technology".Substage := 52; //заполнение газом
               10:
                   "Technology".Substage := 53; //контроль давления перед БГ
               11:
                   "Technology".Substage := 54; //давления перед БГ не в норме. Устраните неисправность. Для продолжения нажмите кн.Розжиг
               12:
                   "Technology".Substage := 55; //проверка давления между ПЗК с открытым КБ
               13:
                   "Technology".Substage := 56; //проверка давления между ПЗК с закрытым КБ
               14:
                   "Technology".Substage := 57; //проверка на MIN. Открытие КО 
               15:
                   "Technology".Substage := 58; //проверка на MIN
               16:
                   "Technology".Substage := 58; //проверка на MIN
               17:
                   "Technology".Substage := 59; //проверка на MAX. Открытие КБ
               18:
                   "Technology".Substage := 59; //проверка на MAX. Открытие КБ
               19:
                   "Technology".Substage := 60; //проверка на MAX. Открытие КО
               20:
                   "Technology".Substage := 61; //проверка на MAX
               21:
                   "Technology".Substage := 62; //проверка на MAX
               22:
                   IF "Message".PRESS_not_initial_state_gas THEN
                       "Technology".Substage := 63; //Механизмы по газу не переведены в исходное состояние. Устраните неисправность и для продолжения нажмите кн.Розжиг
                   END_IF;
                   IF "Message".PRESS_PZK1_or_KO_untight THEN
                       "Technology".Substage := 64; //ПЗК1 или КО неплотен. Устраните неисправность и для продолжения нажмите кн.Розжиг
                   END_IF;
                   IF "Message".PRESS_Not_orifice_plate_or_PZK1_untight THEN
                       "Technology".Substage := 65; //нет дроссельной шайбы или ПЗК1 неплотен. Устраните неисправность и для продолжения нажмите кн.Розжиг
                   END_IF;
                   IF "Message".PRESS_PZK2_or_KB_untight THEN
                       "Technology".Substage := 66; //ПЗК2 или КБ неплотен. Устраните неисправность и для продолжения нажмите кн.Розжиг
                   END_IF;
               23:
                   "Technology".Substage := 175; //опрессовка успешно проведена
               ELSE
                   "Technology".Substage := 0; //неизвестно
           END_CASE;
       5:  //розжиг
           "HMI".INDICATION_TIME_1 := 255;
           "HMI".INDICATION_TIME_2 := 255;
           CASE "Technology".Regim_ignition_step OF
               0:
                   IF NOT "Message".IGNITION_ZRG_not_close THEN
                       "Technology".Substage := 70; //закрываем ЗРГ
                   ELSE
                       "Technology".Substage := 71; //ЗРГ не закрылся
                   END_IF;
               1:
                   IF NOT "Message".IGNITION_PZK2_not_close THEN
                       "Technology".Substage := 72; //контроль закрытого положения ПЗК2
                   ELSE
                       "Technology".Substage := 73; //ПЗК2 не закрыт
                   END_IF;
               2:
                   IF NOT "Message".IGNITION_KZ_not_close THEN
                       "Technology".Substage := 74; //контроль закрытого положения КЗ
                   ELSE
                       "Technology".Substage := 75; //КЗ не закрыт
                   END_IF;
               3:
                   IF NOT "Message".IGNITION_KB_not_close THEN
                       "Technology".Substage := 76; //закрываем КБ
                   ELSE
                       "Technology".Substage := 77; //КБ не закрылся
                   END_IF;
               4:
                   "Technology".Substage := 76; //закрываем КБ
               5:
                   IF NOT "Message".IGNITION_PZK1_not_open THEN
                       "Technology".Substage := 78; //открываем ПЗК1
                   ELSE
                       "Technology".Substage := 79; //ПЗК1 не открылся
                   END_IF;

               6:
                   "Technology".Substage := 78; //открываем ПЗК1
               7:
                   "Technology".Substage := 80; //включаем ИВН
               8:
                   IF "Technology".CNT_Igniter = 1 THEN
                       "Technology".Substage := 81; //включаем ИВН. 1 попытка розжига запальника
                   END_IF;
                   IF "Technology".CNT_Igniter = 2 THEN
                       "Technology".Substage := 82; //включаем ИВН. 2 попытка розжига запальника
                   END_IF;
               9:
                   IF "Technology".CNT_Igniter = 1 THEN
                       IF NOT "Message".IGNITION_KZ_not_open THEN
                           "Technology".Substage := 83; //открываем КЗ. 1 попытка розжига запальника
                       ELSE
                           "Technology".Substage := 84; //КЗ не открылся. 1 попытка розжига запальника
                       END_IF;
                   END_IF;
                   IF "Technology".CNT_Igniter = 2 THEN
                       IF NOT "Message".IGNITION_KZ_not_open THEN
                           "Technology".Substage := 85; //открываем КЗ. 2 попытка розжига запальника
                       ELSE
                           "Technology".Substage := 86; //КЗ не открылся. 2 попытка розжига запальника
                       END_IF;
                   END_IF;
               10:
                   IF "Technology".CNT_Igniter = 1 THEN
                       "Technology".Substage := 87; //розжиг запальника 1 попытка
                   END_IF;
                   IF "Technology".CNT_Igniter = 2 THEN
                       "Technology".Substage := 88; //розжиг запальника 2 попытка
                   END_IF;
               11:
                   IF "Technology".CNT_Igniter = 1 THEN
                       "Technology".Substage := 89; //контроль пламени запальника. 1 попытка розжига
                   END_IF;
                   IF "Technology".CNT_Igniter = 2 THEN
                       "Technology".Substage := 90; //контроль пламени запальника. 2 попытка розжига
                   END_IF;
               12:
                   "Technology".Substage := 91; //запальник не разжегся. Перевод клапанов в исходное положение
               13:
                   IF NOT "Message".IGNITION_not_initial_state_gas THEN
                       "Technology".Substage := 92; //запальник не разжегся. Для повторной попытки нажмите кн. РОЗЖИГ
                   ELSE
                       "Technology".Substage := 93; //газовые клапана не переведены в исходное состояние
                   END_IF;
               14:
                   "Technology".Substage := 94; //открываем ПЗК2
               15:
                   "Technology".Substage := 95; //розжиг горелки
               16:
                   "Technology".Substage := 96; //розжиг горелки
               17:
                   "Technology".Substage := 97; //стабилизация пламени горелки
               18:
                   IF "KZ_control_open".Value THEN
                       "Technology".Substage := 98; //ожидание закрытия КЗ
                   ELSE
                       IF "Message".TEST_IGNITION_ok THEN
                           "Technology".Substage := 99; //тестовый розжиг успешно произведен
                       END_IF;
                   END_IF;
               19:
                   "Technology".Substage := 100; //режим ручного розжига
               20:
                   "Technology".Substage := 88; //розжиг запальника 2 попытка
               21:
                   "Technology".Substage := 88; //розжиг запальника 2 попытка
               ELSE
                   "Technology".Substage := 0; //неизвестно
           END_CASE;
       6:  //выход на MIN мощность
           "HMI".INDICATION_TIME_1 := 255;
           "HMI".INDICATION_TIME_2 := 255;
           CASE "Technology".Regim_min_power_step OF
               0:
                   "Technology".Substage := 110; //переводим ПИД разряжения на работу по режимной карте
               1:
                   "Technology".Substage := 111; //переводим ПИД разряжения на работу по режимной карте
               2:
                   "Technology".Substage := 112; //переводим ПИД давления воздуха на работу по режимной карте
               3:
                   "Technology".Substage := 113; //переводим ПИД давления воздуха на работу по режимной карте
               4:
                   "Technology".Substage := 114; //открываем ЗРГ до значения минимальной мощности
               ELSE
                   "Technology".Substage := 0; //неизвестно
           END_CASE;
       7:  //прогрев
           CASE "Technology".Regim_heating_step OF
               0:
                   "HMI".INDICATION_TIME_1 := 255;
                   "HMI".INDICATION_TIME_2 := 255;
                   "Technology".Substage := 115; //переводим ЗРГ в дистанционный режим
               1:
                   "HMI".TIME_converter_IN := "Timer_HEATING_temp_DB".PT - "Timer_HEATING_temp_DB".ET;
                   "HMI".INDICATION_TIME_1 := INT_TO_USINT("HMI".TIME_converter_minute);
                   "HMI".INDICATION_TIME_2 := INT_TO_USINT("HMI".TIME_converter_second);

